KUKA KRL program: MyProgram_037().src

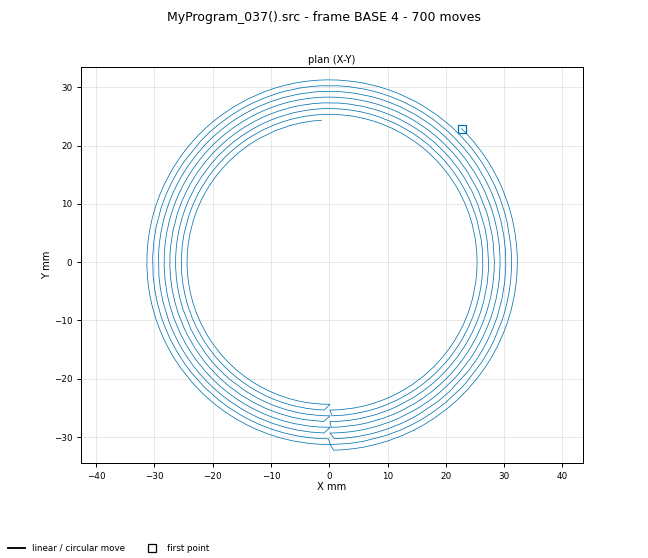
[picture p0: tool path of MyProgram_037().src in frame BASE 4, 700 of 700 moves have a stored position in this frame; points joined in program order, loops and branches not executed]
&ACCESS RVP
&REL 1
&PARAM TEMPLATE = C:\KRC\Roboter\Template\vorgabe
&PARAM EDITMASK = *
DEF MyProgram_037()
; ---- Setting reference (Base) ----
$BASE = BASE_DATA[4]

; --------------------------
; ---- Setting tool (TCP) ----
$TOOL = TOOL_DATA[3]
; --------------------------

$VEL.CP = VEL_APROX_PRINT
Startdeposition()
$VEL.CP = VEL_PRINT
LIN {X 22.7221,Y 22.9099,Z 61,A 36.8926,B 24.82,C -3.0943,E1 25.1146,E2 -314.0122} C_DIS
LIN {X 23.9604,Y 21.6116,Z 61,A 34.1206,B 24.8202,C -3.0927,E1 25.1199,E2 -311.2486} C_DIS
LIN {X 24.912,Y 20.5075,Z 61,A 31.2026,B 24.8214,C -3.0826,E1 25.1251,E2 -308.3199} C_DIS
LIN {X 26.1407,Y 18.916,Z 61,A 27.904,B 24.8219,C -3.0777,E1 25.1306,E2 -305.0254} C_DIS
LIN {X 27.166,Y 17.4114,Z 61,A 24.6548,B 24.8229,C -3.0694,E1 25.1357,E2 -301.7727} C_DIS
LIN {X 28.0132,Y 16.0124,Z 61,A 21.6335,B 24.8239,C -3.0603,E1 25.1399,E2 -298.7454} C_DIS
LIN {X 29.0213,Y 14.1043,Z 61,A 17.6844,B 24.8253,C -3.0484,E1 25.1449,E2 -294.7892} C_DIS
LIN {X 29.7593,Y 12.4714,Z 61,A 14.5862,B 24.8262,C -3.0407,E1 25.1484,E2 -291.6895} C_DIS
LIN {X 30.8171,Y 9.5631,Z 61,A 8.5757,B 24.8288,C -3.0179,E1 25.1538,E2 -285.6589} C_DIS
LIN {X 31.4239,Y 7.3275,Z 61,A 5.4377,B 24.8287,C -3.0189,E1 25.1559,E2 -282.5414} C_DIS
LIN {X 31.8366,Y 5.2519,Z 61,A 0.8875,B 24.8312,C -2.9966,E1 25.1582,E2 -277.9651} C_DIS
LIN {X 32.1427,Y 2.8314,Z 61,A -2.7277,B 24.8316,C -2.9931,E1 25.1593,E2 -274.363} C_DIS
LIN {X 32.236,Y 1.4111,Z 61,A -5.1666,B 24.8324,C -2.9865,E1 25.1597,E2 -271.9229} C_DIS
LIN {X 32.266,Y -0.0088,Z 61,A -7.9428,B 24.8337,C -2.9751,E1 25.1597,E2 -269.1363} C_DIS
LIN {X 32.2046,Y -2.0098,Z 61,A -11.4053,B 24.8348,C -2.9652,E1 25.1593,E2 -265.6709} C_DIS
LIN {X 32.0309,Y -3.8974,Z 61,A -14.9413,B 24.8362,C -2.9523,E1 25.1583,E2 -262.1254} C_DIS
LIN {X 31.7367,Y -5.8263,Z 61,A -18.1738,B 24.837,C -2.9447,E1 25.1568,E2 -258.8938} C_DIS
LIN {X 31.2216,Y -8.147,Z 61,A -22.8563,B 24.8392,C -2.9253,E1 25.1537,E2 -254.1926} C_DIS
LIN {X 30.6383,Y -10.1233,Z 61,A -25.8233,B 24.8394,C -2.9237,E1 25.1512,E2 -251.2384} C_DIS
LIN {X 29.8919,Y -12.1501,Z 61,A -30.2718,B 24.8416,C -2.9038,E1 25.1467,E2 -246.7676} C_DIS
LIN {X 28.8147,Y -14.5215,Z 61,A -34.7253,B 24.8428,C -2.8926,E1 25.1414,E2 -242.3116} C_DIS
LIN {X 27.7798,Y -16.4144,Z 61,A -38.242,B 24.8435,C -2.8861,E1 25.1365,E2 -238.7975} C_DIS
LIN {X 26.8232,Y -17.9358,Z 61,A -41.3536,B 24.8443,C -2.8784,E1 25.1318,E2 -235.6833} C_DIS
LIN {X 25.4842,Y -19.7918,Z 61,A -45.8741,B 24.8462,C -2.8616,E1 25.1242,E2 -231.1447} C_DIS
LIN {X 23.7816,Y -21.8079,Z 61,A -50.4062,B 24.8472,C -2.8519,E1 25.1158,E2 -226.61} C_DIS
LIN {X 22.0503,Y -23.5572,Z 61,A -54.7017,B 24.8482,C -2.8426,E1 25.1072,E2 -222.3105} C_DIS
LIN {X 20.232,Y -25.1362,Z 61,A -58.9185,B 24.8491,C -2.8341,E1 25.0982,E2 -218.0897} C_DIS
LIN {X 18.0334,Y -26.7573,Z 61,A -64.2333,B 24.8508,C -2.8186,E1 25.086,E2 -212.7565} C_DIS
LIN {X 16.0936,Y -27.9669,Z 61,A -67.2597,B 24.8502,C -2.8242,E1 25.0788,E2 -209.7528} C_DIS
LIN {X 14.6043,Y -28.7727,Z 61,A -70.6753,B 24.8512,C -2.8141,E1 25.0703,E2 -206.3229} C_DIS
LIN {X 12.6886,Y -29.6677,Z 61,A -74.4308,B 24.8518,C -2.8085,E1 25.0608,E2 -202.5634} C_DIS
LIN {X 10.2156,Y -30.6072,Z 61,A -79.763,B 24.8532,C -2.7951,E1 25.0467,E2 -197.2101} C_DIS
LIN {X 7.7675,Y -31.3182,Z 61,A -83.5174,B 24.8528,C -2.7994,E1 25.0366,E2 -193.472} C_DIS
LIN {X 6.0925,Y -31.6861,Z 61,A -86.5057,B 24.853,C -2.7975,E1 25.0284,E2 -190.4828} C_DIS
LIN {X 4.35,Y -31.9726,Z 61,A -89.6463,B 24.8532,C -2.7953,E1 25.0197,E2 -187.3398} C_DIS
LIN {X 2.5855,Y -32.1631,Z 61,A -92.4941,B 24.853,C -2.797,E1 25.0118,E2 -184.4979} C_DIS
LIN {X 0.7515,Y -32.2571,Z 61,A -95.8832,B 24.8533,C -2.7944,E1 25.0024,E2 -181.1037} C_DIS
LIN {X 0.7515,Y -32.2571,Z 61,A -95.8832,B 24.8533,C -2.7944,E1 25.0024,E2 -181.1037} C_DIS
Enddeposition()
LIN {X 0.1793,Y -31.277,Z 61,A -95.2426,B 24.8496,C -2.8293,E1 25.0044,E2 -181.8273} C_DIS
Startdeposition()
$VEL.CP = VEL_PRINT
LIN {X 3.3211,Y -31.1043,Z 61,A -89.5129,B 24.8494,C -2.8315,E1 25.0204,E2 -187.5594} C_DIS
LIN {X 5.8203,Y -30.7348,Z 61,A -84.3877,B 24.8484,C -2.8408,E1 25.0345,E2 -192.7011} C_DIS
LIN {X 9.7861,Y -29.7112,Z 61,A -76.8094,B 24.8474,C -2.8498,E1 25.0548,E2 -200.288} C_DIS
LIN {X 12.2324,Y -28.7911,Z 61,A -73.017,B 24.848,C -2.8443,E1 25.0646,E2 -204.0588} C_DIS
LIN {X 13.9421,Y -28.0031,Z 61,A -69.1318,B 24.8469,C -2.855,E1 25.0744,E2 -207.9593} C_DIS
LIN {X 15.7865,Y -27.0066,Z 61,A -66.0402,B 24.8471,C -2.8524,E1 25.0819,E2 -211.0355} C_DIS
LIN {X 17.661,Y -25.8198,Z 61,A -60.7635,B 24.8447,C -2.8754,E1 25.0943,E2 -216.3493} C_DIS
LIN {X 19.9043,Y -24.1326,Z 61,A -55.5619,B 24.8434,C -2.8872,E1 25.1057,E2 -221.5593} C_DIS
LIN {X 22.7108,Y -21.5119,Z 61,A -49.7962,B 24.8434,C -2.887,E1 25.1171,E2 -227.3007} C_DIS
LIN {X 23.4756,Y -20.6753,Z 61,A -46.3418,B 24.8408,C -2.9105,E1 25.1236,E2 -230.795} C_DIS
LIN {X 26.1964,Y -17.0974,Z 61,A -38.73,B 24.8393,C -2.924,E1 25.1359,E2 -238.4019} C_DIS
LIN {X 27.5194,Y -14.8741,Z 61,A -34.5181,B 24.8386,C -2.9303,E1 25.1417,E2 -242.6068} C_DIS
LIN {X 28.3302,Y -13.2648,Z 61,A -30.4988,B 24.8365,C -2.9497,E1 25.1466,E2 -246.6505} C_DIS
LIN {X 29.6792,Y -9.8843,Z 61,A -24.9159,B 24.8359,C -2.9548,E1 25.1521,E2 -252.2145} C_DIS
LIN {X 30.0713,Y -8.6185,Z 61,A -22.3462,B 24.8349,C -2.9642,E1 25.1541,E2 -254.7917} C_DIS
LIN {X 30.4929,Y -6.9814,Z 61,A -19.0418,B 24.8335,C -2.9766,E1 25.1563,E2 -258.1064} C_DIS
LIN {X 30.8584,Y -5.1295,Z 61,A -15.6608,B 24.8324,C -2.9864,E1 25.158,E2 -261.4906} C_DIS
LIN {X 31.1322,Y -3.0618,Z 61,A -11.7675,B 24.8309,C -2.9993,E1 25.1593,E2 -265.3916} C_DIS
LIN {X 31.2639,Y -1.0643,Z 61,A -8.2104,B 24.8298,C -3.0093,E1 25.1597,E2 -268.9512} C_DIS
LIN {X 31.2659,Y 0.9986,Z 61,A -4.0775,B 24.8279,C -3.026,E1 25.1595,E2 -273.099} C_DIS
LIN {X 31.1526,Y 2.8404,Z 61,A -0.0947,B 24.8257,C -3.0448,E1 25.1585,E2 -277.1027} C_DIS
LIN {X 30.502,Y 6.9419,Z 61,A 6.4981,B 24.8247,C -3.0539,E1 25.1552,E2 -283.6785} C_DIS
LIN {X 30.1115,Y 8.4753,Z 61,A 9.5892,B 24.8234,C -3.0651,E1 25.1529,E2 -286.7783} C_DIS
LIN {X 29.2983,Y 10.9626,Z 61,A 13.7921,B 24.8227,C -3.0709,E1 25.1491,E2 -290.9715} C_DIS
LIN {X 28.4168,Y 13.078,Z 61,A 18.7309,B 24.8202,C -3.0925,E1 25.1436,E2 -295.9345} C_DIS
LIN {X 27.2863,Y 15.2975,Z 61,A 22.9812,B 24.8193,C -3.1005,E1 25.138,E2 -300.1813} C_DIS
LIN {X 26.2057,Y 17.0833,Z 61,A 26.3044,B 24.8189,C -3.1036,E1 25.1331,E2 -303.4952} C_DIS
LIN {X 25.2575,Y 18.4557,Z 61,A 29.3022,B 24.8181,C -3.1103,E1 25.1282,E2 -306.4942} C_DIS
LIN {X 24.5119,Y 19.4351,Z 61,A 31.6052,B 24.8174,C -3.1163,E1 25.1243,E2 -308.8004} C_DIS
LIN {X 23.7173,Y 20.3976,Z 61,A 34.2425,B 24.8163,C -3.1259,E1 25.1195,E2 -311.4486} C_DIS
LIN {X 22.3374,Y 21.899,Z 61,A 37.6321,B 24.8159,C -3.1295,E1 25.113,E2 -314.8319} C_DIS
LIN {X 21.2569,Y 22.9504,Z 61,A 40.4087,B 24.8152,C -3.1352,E1 25.1074,E2 -317.6107} C_DIS
LIN {X 20.2008,Y 23.8849,Z 61,A 43.3561,B 24.8141,C -3.1446,E1 25.1011,E2 -320.5688} C_DIS
LIN {X 18.523,Y 25.2082,Z 61,A 47.5292,B 24.8129,C -3.1545,E1 25.0918,E2 -324.7504} C_DIS
LIN {X 15.977,Y 26.894,Z 61,A 52.4422,B 24.8129,C -3.1548,E1 25.0803,E2 -329.6481} C_DIS
LIN {X 14.9451,Y 27.4809,Z 61,A 55.3612,B 24.8115,C -3.1665,E1 25.0731,E2 -332.5865} C_DIS
LIN {X 12.1463,Y 28.8274,Z 61,A 60.2984,B 24.8117,C -3.1641,E1 25.0606,E2 -337.5056} C_DIS
LIN {X 10.3203,Y 29.5304,Z 61,A 64.2509,B 24.8109,C -3.1715,E1 25.0502,E2 -341.4674} C_DIS
LIN {X 8.4349,Y 30.123,Z 61,A 68.0075,B 24.8104,C -3.1755,E1 25.0401,E2 -345.2271} C_DIS
LIN {X 5.8555,Y 30.729,Z 61,A 72.4111,B 24.8107,C -3.1729,E1 25.0281,E2 -349.6186} C_DIS
LIN {X 4.2839,Y 30.987,Z 61,A 75.855,B 24.8099,C -3.1793,E1 25.0186,E2 -353.0747} C_DIS
LIN {X 1.5654,Y 31.243,Z 61,A 80.5109,B 24.8103,C -3.1759,E1 25.0057,E2 -357.7202} C_DIS
LIN {X -0.4527,Y 31.2782,Z 61,A 83.939,B 24.8107,C -3.1724,E1 24.9961,E2 -361.14} C_DIS
LIN {X -1.9504,Y 31.2214,Z 61,A 86.8625,B 24.8107,C -3.1733,E1 24.988,E2 -364.0661} C_DIS
LIN {X -3.7004,Y 31.0622,Z 61,A 89.7933,B 24.8112,C -3.1688,E1 24.9798,E2 -366.9879} C_DIS
LIN {X -4.8807,Y 30.8989,Z 61,A 92.0557,B 24.8112,C -3.1681,E1 24.9736,E2 -369.2507} C_DIS
LIN {X -6.0959,Y 30.6823,Z 61,A 94.5824,B 24.8112,C -3.1689,E1 24.9666,E2 -371.7821} C_DIS
LIN {X -7.8851,Y 30.2715,Z 61,A 97.7613,B 24.8117,C -3.1641,E1 24.958,E2 -374.9538} C_DIS
LIN {X -9.34,Y 29.855,Z 61,A 100.6774,B 24.8119,C -3.1624,E1 24.9502,E2 -377.8709} C_DIS
LIN {X -10.9576,Y 29.3002,Z 61,A 104.3444,B 24.8119,C -3.1635,E1 24.9406,E2 -381.5478} C_DIS
LIN {X -13.786,Y 28.0804,Z 61,A 109.2809,B 24.8136,C -3.1489,E1 24.9281,E2 -386.4614} C_DIS
LIN {X -16.3147,Y 26.6903,Z 61,A 115.7502,B 24.8134,C -3.1501,E1 24.9124,E2 -392.9529} C_DIS
LIN {X -18.6587,Y 25.1078,Z 61,A 120.0777,B 24.8155,C -3.1326,E1 24.9026,E2 -397.2535} C_DIS
LIN {X -20.009,Y 24.0456,Z 61,A 123.0586,B 24.8164,C -3.1246,E1 24.8962,E2 -400.2265} C_DIS
LIN {X -21.1218,Y 23.0743,Z 61,A 125.7069,B 24.8172,C -3.1181,E1 24.8907,E2 -402.8698} C_DIS
LIN {X -22.43,Y 21.8051,Z 61,A 129.3952,B 24.8178,C -3.1131,E1 24.8834,E2 -406.5617} C_DIS
LIN {X -24.1295,Y 19.9081,Z 61,A 134.5719,B 24.8187,C -3.1056,E1 24.874,E2 -411.7439} C_DIS
LIN {X -25.5591,Y 18.0363,Z 61,A 138.1819,B 24.8206,C -3.0887,E1 24.868,E2 -415.331} C_DIS
LIN {X -26.9094,Y 15.9512,Z 61,A 143.7462,B 24.8212,C -3.084,E1 24.8598,E2 -420.9126} C_DIS
LIN {X -28.2304,Y 13.4761,Z 61,A 148.1193,B 24.8236,C -3.0633,E1 24.8544,E2 -425.2597} C_DIS
LIN {X -29.0622,Y 11.5738,Z 61,A 151.9664,B 24.8249,C -3.0524,E1 24.8502,E2 -429.102} C_DIS
LIN {X -29.7747,Y 9.5928,Z 61,A 156.0479,B 24.826,C -3.0425,E1 24.8466,E2 -433.1829} C_DIS
LIN {X -30.3453,Y 7.5996,Z 61,A 159.7045,B 24.8275,C -3.0298,E1 24.844,E2 -436.8303} C_DIS
LIN {X -30.7795,Y 5.5835,Z 61,A 163.4375,B 24.8288,C -3.0178,E1 24.8419,E2 -440.5566} C_DIS
LIN {X -31.0699,Y 3.635,Z 61,A 167.201,B 24.83,C -3.0076,E1 24.8406,E2 -444.3184} C_DIS
LIN {X -31.2361,Y 1.691,Z 61,A 170.4385,B 24.8315,C -2.994,E1 24.8399,E2 -447.5426} C_DIS
LIN {X -31.2747,Y -0.673,Z 61,A 175.5679,B 24.8324,C -2.9864,E1 24.8399,E2 -452.6848} C_DIS
LIN {X -31.1425,Y -2.9504,Z 61,A 179.1206,B 24.8344,C -2.9688,E1 24.8407,E2 -456.2167} C_DIS
LIN {X -30.9732,Y -4.3828,Z 61,A -178.3923,B 24.8354,C -2.9596,E1 24.8416,E2 -458.6965} C_DIS
LIN {X -30.7489,Y -5.7508,Z 61,A -175.6308,B 24.8361,C -2.9535,E1 24.8429,E2 -461.4599} C_DIS
LIN {X -30.3552,Y -7.5574,Z 61,A -172.6642,B 24.8375,C -2.9402,E1 24.8448,E2 -464.4121} C_DIS
LIN {X -29.7953,Y -9.529,Z 61,A -167.6721,B 24.8377,C -2.9386,E1 24.8488,E2 -469.4292} C_DIS
LIN {X -29.0107,Y -11.7023,Z 61,A -164.0836,B 24.8396,C -2.9217,E1 24.8524,E2 -472.9972} C_DIS
LIN {X -28.2977,Y -13.333,Z 61,A -160.8621,B 24.8406,C -2.9124,E1 24.8561,E2 -476.2141} C_DIS
LIN {X -27.3621,Y -15.1617,Z 61,A -157.5041,B 24.8421,C -2.8992,E1 24.8605,E2 -479.5584} C_DIS
LIN {X -26.5372,Y -16.5628,Z 61,A -153.809,B 24.8423,C -2.8973,E1 24.8659,E2 -483.2679} C_DIS
LIN {X -25.4676,Y -18.1646,Z 61,A -149.9018,B 24.8429,C -2.8918,E1 24.8721,E2 -487.1813} C_DIS
LIN {X -23.4143,Y -20.7446,Z 61,A -144.5543,B 24.845,C -2.8724,E1 24.8816,E2 -492.5069} C_DIS
LIN {X -21.7484,Y -22.4847,Z 61,A -139.595,B 24.8455,C -2.8679,E1 24.8914,E2 -497.4768} C_DIS
LIN {X -19.7938,Y -24.2225,Z 61,A -134.708,B 24.8463,C -2.8599,E1 24.9018,E2 -502.3635} C_DIS
LIN {X -17.9022,Y -25.6528,Z 61,A -131.385,B 24.8481,C -2.8435,E1 24.9092,E2 -505.6591} C_DIS
LIN {X -16.1813,Y -26.7715,Z 61,A -126.5019,B 24.8476,C -2.8482,E1 24.9208,E2 -510.5689} C_DIS
LIN {X -14.1331,Y -27.9074,Z 61,A -122.7805,B 24.8487,C -2.8375,E1 24.9299,E2 -514.275} C_DIS
LIN {X -12.3744,Y -28.7304,Z 61,A -119.0798,B 24.849,C -2.835,E1 24.9394,E2 -517.9789} C_DIS
LIN {X -10.1671,Y -29.5837,Z 61,A -114.3689,B 24.849,C -2.835,E1 24.9518,E2 -522.6992} C_DIS
LIN {X -8.2154,Y -30.1838,Z 61,A -111.3645,B 24.8501,C -2.8252,E1 24.9598,E2 -525.6852} C_DIS
LIN {X -6.0483,Y -30.6918,Z 61,A -106.3449,B 24.8492,C -2.8331,E1 24.9735,E2 -530.7296} C_DIS
LIN {X -3.3817,Y -31.0983,Z 61,A -101.8901,B 24.8499,C -2.8271,E1 24.9858,E2 -535.1734} C_DIS
LIN {X -1.2466,Y -31.2571,Z 61,A -97.8183,B 24.8497,C -2.8289,E1 24.9972,E2 -539.2508} C_DIS
LIN {X 0.1793,Y -31.277,Z 61,A -95.2424,B 24.8497,C -2.8292,E1 25.0044,E2 -541.8272} C_DIS
Enddeposition()
LIN {X 0.1793,Y -31.277,Z 61,A -95.2424,B 24.8497,C -2.8292,E1 25.0044,E2 -541.8272} C_DIS
Startdeposition()
$VEL.CP = VEL_PRINT
LIN {X -0.1083,Y -30.2967,Z 61,A -97.7907,B 24.8501,C -2.8248,E1 24.9973,E2 -539.2685} C_DIS
LIN {X -1.7664,Y -30.2454,Z 61,A -100.7174,B 24.8499,C -2.8266,E1 24.9891,E2 -536.3455} C_DIS
LIN {X -3.5776,Y -30.0849,Z 61,A -104.4761,B 24.8502,C -2.8238,E1 24.9786,E2 -532.5779} C_DIS
LIN {X -5.7242,Y -29.7511,Z 61,A -108.6372,B 24.8502,C -2.8245,E1 24.9672,E2 -528.4145} C_DIS
LIN {X -7.9,Y -29.2487,Z 61,A -112.9088,B 24.8499,C -2.8264,E1 24.9556,E2 -524.1412} C_DIS
LIN {X -9.8571,Y -28.6489,Z 61,A -116.5327,B 24.8494,C -2.8315,E1 24.946,E2 -520.523} C_DIS
LIN {X -12.0715,Y -27.7881,Z 61,A -121.794,B 24.8496,C -2.8291,E1 24.9324,E2 -515.2441} C_DIS
LIN {X -14.1119,Y -26.8095,Z 61,A -125.1264,B 24.8482,C -2.8425,E1 24.9241,E2 -511.9348} C_DIS
LIN {X -15.2026,Y -26.2056,Z 61,A -127.7329,B 24.8481,C -2.8436,E1 24.9178,E2 -509.3231} C_DIS
LIN {X -17.2127,Y -24.9324,Z 61,A -132.0881,B 24.8472,C -2.8516,E1 24.9076,E2 -504.973} C_DIS
LIN {X -18.9208,Y -23.6626,Z 61,A -136.9417,B 24.8472,C -2.8518,E1 24.8969,E2 -500.1021} C_DIS
LIN {X -21.3596,Y -21.4865,Z 61,A -143.2342,B 24.846,C -2.8632,E1 24.8841,E2 -493.811} C_DIS
LIN {X -23.5988,Y -19.0001,Z 61,A -149.3266,B 24.8443,C -2.8791,E1 24.8731,E2 -487.729} C_DIS
LIN {X -24.7571,Y -17.4644,Z 61,A -152.8937,B 24.8432,C -2.8884,E1 24.8672,E2 -484.1666} C_DIS
LIN {X -26.1364,Y -15.323,Z 61,A -157.5379,B 24.8418,C -2.9019,E1 24.8604,E2 -479.5311} C_DIS
LIN {X -27.4184,Y -12.8894,Z 61,A -163.2384,B 24.8406,C -2.9124,E1 24.8533,E2 -473.8249} C_DIS
LIN {X -28.2493,Y -10.9495,Z 61,A -166.6876,B 24.839,C -2.9274,E1 24.8497,E2 -470.3925} C_DIS
LIN {X -28.8492,Y -9.2519,Z 61,A -170.1049,B 24.8379,C -2.9372,E1 24.8467,E2 -466.979} C_DIS
LIN {X -29.4938,Y -6.9298,Z 61,A -174.3156,B 24.8361,C -2.9531,E1 24.8437,E2 -462.7818} C_DIS
LIN {X -29.9388,Y -4.644,Z 61,A -179.87,B 24.8355,C -2.9587,E1 24.841,E2 -457.2079} C_DIS
LIN {X -30.1985,Y -2.439,Z 61,A 175.975,B 24.834,C -2.9719,E1 24.84,E2 -453.0596} C_DIS
LIN {X -30.2834,Y 0.8875,Z 61,A 170.1741,B 24.8314,C -2.9948,E1 24.84,E2 -447.2787} C_DIS
LIN {X -30.0832,Y 3.5884,Z 61,A 164.9418,B 24.8297,C -3.0101,E1 24.8413,E2 -442.0516} C_DIS
LIN {X -29.6827,Y 6.0689,Z 61,A 159.6211,B 24.8284,C -3.0211,E1 24.844,E2 -436.7256} C_DIS
LIN {X -28.8326,Y 9.3041,Z 61,A 153.6942,B 24.8259,C -3.0431,E1 24.8486,E2 -430.8171} C_DIS
LIN {X -28.0084,Y 11.5504,Z 61,A 149.1158,B 24.8244,C -3.0562,E1 24.8533,E2 -426.2445} C_DIS
LIN {X -27.0518,Y 13.6423,Z 61,A 145.6235,B 24.8223,C -3.0748,E1 24.8574,E2 -422.7777} C_DIS
LIN {X -26.0575,Y 15.4565,Z 61,A 140.2107,B 24.8223,C -3.0753,E1 24.8649,E2 -417.3379} C_DIS
LIN {X -24.8873,Y 17.2777,Z 61,A 135.6577,B 24.8213,C -3.083,E1 24.8722,E2 -412.781} C_DIS
LIN {X -21.994,Y 20.8368,Z 61,A 128.3614,B 24.8176,C -3.1147,E1 24.8854,E2 -405.5272} C_DIS
LIN {X -20.6237,Y 22.1937,Z 61,A 124.5732,B 24.8167,C -3.122,E1 24.893,E2 -401.7408} C_DIS
LIN {X -19.0927,Y 23.5236,Z 61,A 120.2867,B 24.8162,C -3.1268,E1 24.9022,E2 -397.4494} C_DIS
LIN {X -17.0972,Y 25.0118,Z 61,A 116.1796,B 24.8145,C -3.1408,E1 24.9115,E2 -393.3615} C_DIS
LIN {X -15.5028,Y 26.0301,Z 61,A 112.0706,B 24.8143,C -3.143,E1 24.9212,E2 -389.2449} C_DIS
LIN {X -13.5594,Y 27.0934,Z 61,A 107.8903,B 24.8134,C -3.1498,E1 24.9316,E2 -385.0695} C_DIS
LIN {X -11.1624,Y 28.1657,Z 61,A 102.7878,B 24.8128,C -3.1556,E1 24.9447,E2 -379.969} C_DIS
LIN {X -8.6144,Y 29.0463,Z 61,A 98.1678,B 24.8116,C -3.1656,E1 24.9569,E2 -375.3644} C_DIS
LIN {X -7.4328,Y 29.3704,Z 61,A 95.5053,B 24.8116,C -3.1647,E1 24.9642,E2 -372.6961} C_DIS
LIN {X -5.0851,Y 29.8671,Z 61,A 91.1536,B 24.811,C -3.1699,E1 24.9761,E2 -368.3521} C_DIS
LIN {X -2.8898,Y 30.1588,Z 61,A 86.9107,B 24.8108,C -3.1717,E1 24.9878,E2 -364.1107} C_DIS
LIN {X -1.489,Y 30.2599,Z 61,A 83.7084,B 24.8113,C -3.1675,E1 24.9968,E2 -360.8976} C_DIS
LIN {X 1.7595,Y 30.2458,Z 61,A 78.3913,B 24.8103,C -3.1762,E1 25.0116,E2 -355.6022} C_DIS
LIN {X 3.3881,Y 30.1066,Z 61,A 74.7935,B 24.8109,C -3.1708,E1 25.0216,E2 -351.9938} C_DIS
LIN {X 6.0588,Y 29.6848,Z 61,A 70.2105,B 24.8105,C -3.1744,E1 25.0342,E2 -347.4243} C_DIS
LIN {X 7.6214,Y 29.3225,Z 61,A 67.3022,B 24.8105,C -3.1741,E1 25.042,E2 -344.5194} C_DIS
LIN {X 8.8433,Y 28.9774,Z 61,A 64.8089,B 24.8109,C -3.1714,E1 25.0487,E2 -342.0241} C_DIS
LIN {X 10.5374,Y 28.4057,Z 61,A 61.2512,B 24.8114,C -3.1666,E1 25.0581,E2 -338.4622} C_DIS
LIN {X 12.6517,Y 27.5291,Z 61,A 56.5705,B 24.8124,C -3.1582,E1 25.0701,E2 -333.7727} C_DIS
LIN {X 14.7691,Y 26.4532,Z 61,A 52.4965,B 24.8126,C -3.157,E1 25.0801,E2 -329.7076} C_DIS
LIN {X 15.97,Y 25.7457,Z 61,A 49.6207,B 24.8134,C -3.1505,E1 25.087,E2 -326.8252} C_DIS
LIN {X 17.8127,Y 24.5075,Z 61,A 45.2964,B 24.8144,C -3.1422,E1 25.0969,E2 -322.4961} C_DIS
LIN {X 19.9808,Y 22.7742,Z 61,A 40.5699,B 24.8148,C -3.1387,E1 25.107,E2 -317.7793} C_DIS
LIN {X 21.1552,Y 21.687,Z 61,A 37.0416,B 24.8162,C -3.1266,E1 25.1142,E2 -314.2371} C_DIS
LIN {X 23.0143,Y 19.7039,Z 61,A 32.585,B 24.8165,C -3.1237,E1 25.1225,E2 -309.7933} C_DIS
LIN {X 24.2227,Y 18.1978,Z 61,A 28.2223,B 24.8186,C -3.1064,E1 25.13,E2 -305.4102} C_DIS
LIN {X 25.3541,Y 16.5854,Z 61,A 24.1344,B 24.8202,C -3.0927,E1 25.1363,E2 -301.3101} C_DIS
LIN {X 27.0232,Y 13.6987,Z 61,A 18.5921,B 24.821,C -3.0856,E1 25.1438,E2 -295.78} C_DIS
LIN {X 27.9171,Y 11.7698,Z 61,A 14.7622,B 24.822,C -3.0769,E1 25.1481,E2 -291.9502} C_DIS
LIN {X 28.5269,Y 10.2035,Z 61,A 10.9832,B 24.824,C -3.0601,E1 25.1518,E2 -288.1527} C_DIS
LIN {X 29.4353,Y 7.1737,Z 61,A 5.6519,B 24.825,C -3.0508,E1 25.1558,E2 -282.83} C_DIS
LIN {X 29.9505,Y 4.5682,Z 61,A -0.1932,B 24.828,C -3.0249,E1 25.1586,E2 -276.9578} C_DIS
LIN {X 30.2349,Y 1.9385,Z 61,A -4.6467,B 24.829,C -3.0166,E1 25.1596,E2 -272.5109} C_DIS
LIN {X 30.2949,Y -0.3425,Z 61,A -8.9772,B 24.8305,C -3.0029,E1 25.1596,E2 -268.1738} C_DIS
LIN {X 30.124,Y -3.2324,Z 61,A -14.8109,B 24.833,C -2.9811,E1 25.1583,E2 -262.323} C_DIS
LIN {X 29.6574,Y -6.1925,Z 61,A -20.1219,B 24.8344,C -2.9681,E1 25.1557,E2 -257.0124} C_DIS
LIN {X 28.8629,Y -9.211,Z 61,A -24.9574,B 24.8349,C -2.964,E1 25.1521,E2 -252.1948} C_DIS
LIN {X 28.0924,Y -11.3454,Z 61,A -30.7262,B 24.8385,C -2.9319,E1 25.1463,E2 -246.3822} C_DIS
LIN {X 27.0866,Y -13.5732,Z 61,A -34.1792,B 24.8383,C -2.9335,E1 25.1422,E2 -242.9516} C_DIS
LIN {X 26.3833,Y -14.8943,Z 61,A -37.27,B 24.8396,C -2.9221,E1 25.138,E2 -239.8499} C_DIS
LIN {X 25.3403,Y -16.6064,Z 61,A -40.3805,B 24.8397,C -2.9203,E1 25.1334,E2 -236.7509} C_DIS
LIN {X 23.953,Y -18.5514,Z 61,A -46.8407,B 24.8437,C -2.8839,E1 25.1226,E2 -230.2355} C_DIS
LIN {X 20.6747,Y -22.1465,Z 61,A -55.9829,B 24.846,C -2.8628,E1 25.1046,E2 -221.0822} C_DIS
LIN {X 18.623,Y -23.8975,Z 61,A -60.9233,B 24.847,C -2.8539,E1 25.0938,E2 -216.1391} C_DIS
LIN {X 15.2202,Y -26.1966,Z 61,A -67.5031,B 24.847,C -2.8534,E1 25.0784,E2 -209.5794} C_DIS
LIN {X 13.4821,Y -27.1315,Z 61,A -70.9533,B 24.8473,C -2.8506,E1 25.0699,E2 -206.1321} C_DIS
LIN {X 12.1806,Y -27.7404,Z 61,A -73.8495,B 24.848,C -2.8444,E1 25.0625,E2 -203.2286} C_DIS
LIN {X 10.1217,Y -28.5562,Z 61,A -78.4977,B 24.8491,C -2.8337,E1 25.0503,E2 -198.5649} C_DIS
LIN {X 8.3465,Y -29.1245,Z 61,A -81.7097,B 24.8491,C -2.8333,E1 25.0417,E2 -195.3574} C_DIS
LIN {X 6.916,Y -29.4969,Z 61,A -84.6101,B 24.8496,C -2.8295,E1 25.0338,E2 -192.4522} C_DIS
LIN {X 4.7564,Y -29.9211,Z 61,A -88.6328,B 24.8498,C -2.8278,E1 25.0228,E2 -188.4297} C_DIS
LIN {X 2.5826,Y -30.186,Z 61,A -92.4841,B 24.8498,C -2.8285,E1 25.0121,E2 -184.5828} C_DIS
LIN {X 0.8989,Y -30.2834,Z 61,A -95.9394,B 24.8501,C -2.8246,E1 25.0024,E2 -181.1192} C_DIS
LIN {X 0.8989,Y -30.2834,Z 61,A -95.9394,B 24.8501,C -2.8246,E1 25.0024,E2 -181.1192} C_DIS
Enddeposition()
LIN {X 0.148,Y -29.3098,Z 61,A -95.712,B 24.8465,C -2.8581,E1 25.0033,E2 -181.4265} C_DIS
Startdeposition()
$VEL.CP = VEL_PRINT
LIN {X 2.0107,Y -29.2427,Z 61,A -92.0588,B 24.8464,C -2.8596,E1 25.0135,E2 -185.0819} C_DIS
LIN {X 3.7148,Y -29.075,Z 61,A -88.9657,B 24.8464,C -2.8588,E1 25.022,E2 -188.171} C_DIS
LIN {X 4.9608,Y -28.8892,Z 61,A -86.4055,B 24.8461,C -2.8616,E1 25.0291,E2 -190.7354} C_DIS
LIN {X 6.1622,Y -28.6568,Z 61,A -83.7025,B 24.8456,C -2.8671,E1 25.0365,E2 -193.4479} C_DIS
LIN {X 7.9763,Y -28.2057,Z 61,A -79.7952,B 24.8448,C -2.8736,E1 25.0471,E2 -197.3645} C_DIS
LIN {X 10.4914,Y -27.3695,Z 61,A -75.5865,B 24.8453,C -2.8692,E1 25.0581,E2 -201.5543} C_DIS
LIN {X 11.7916,Y -26.8355,Z 61,A -71.1886,B 24.8428,C -2.8921,E1 25.0695,E2 -205.9959} C_DIS
LIN {X 15.0472,Y -25.1549,Z 61,A -64.7391,B 24.8424,C -2.8959,E1 25.0853,E2 -212.4357} C_DIS
LIN {X 17.2957,Y -23.6651,Z 61,A -59.7421,B 24.8417,C -2.9029,E1 25.0967,E2 -217.4323} C_DIS
LIN {X 18.7666,Y -22.5166,Z 61,A -55.493,B 24.84,C -2.9181,E1 25.1059,E2 -221.7013} C_DIS
LIN {X 21.1943,Y -20.2484,Z 61,A -49.8511,B 24.8395,C -2.9227,E1 25.1172,E2 -227.3306} C_DIS
LIN {X 22.3114,Y -19.01,Z 61,A -45.9121,B 24.8376,C -2.9394,E1 25.1244,E2 -231.2913} C_DIS
LIN {X 24.1424,Y -16.623,Z 61,A -40.9595,B 24.8372,C -2.9432,E1 25.1326,E2 -236.2291} C_DIS
LIN {X 24.8001,Y -15.6252,Z 61,A -38.3769,B 24.8361,C -2.9528,E1 25.1365,E2 -238.8214} C_DIS
LIN {X 25.6751,Y -14.1403,Z 61,A -35.035,B 24.8351,C -2.962,E1 25.1412,E2 -242.1677} C_DIS
LIN {X 26.337,Y -12.8674,Z 61,A -32.0159,B 24.8339,C -2.9728,E1 25.1449,E2 -245.1965} C_DIS
LIN {X 27.1667,Y -11.006,Z 61,A -28.3627,B 24.8331,C -2.9804,E1 25.1489,E2 -248.8475} C_DIS
LIN {X 27.762,Y -9.4049,Z 61,A -25.2808,B 24.8323,C -2.9871,E1 25.1518,E2 -251.928} C_DIS
LIN {X 28.1054,Y -8.3226,Z 61,A -22.5879,B 24.8308,C -3,E1 25.154,E2 -254.6362} C_DIS
LIN {X 28.6095,Y -6.377,Z 61,A -18.7112,B 24.8295,C -3.0115,E1 25.1566,E2 -258.5176} C_DIS
LIN {X 29.0038,Y -4.2385,Z 61,A -14.659,B 24.8283,C -3.0221,E1 25.1584,E2 -262.5712} C_DIS
LIN {X 29.2053,Y -2.5002,Z 61,A -11.0811,B 24.8269,C -3.0349,E1 25.1594,E2 -266.1581} C_DIS
LIN {X 29.3074,Y -0.5096,Z 61,A -7.4417,B 24.8259,C -3.0437,E1 25.1598,E2 -269.7969} C_DIS
LIN {X 29.2938,Y 1.0136,Z 61,A -4.2793,B 24.8245,C -3.0554,E1 25.1596,E2 -272.9681} C_DIS
LIN {X 29.1565,Y 3.0136,Z 61,A -0.1704,B 24.8228,C -3.07,E1 25.1585,E2 -277.0872} C_DIS
LIN {X 28.7926,Y 5.4913,Z 61,A 4.4077,B 24.8216,C -3.0808,E1 25.1565,E2 -281.664} C_DIS
LIN {X 28.3607,Y 7.4071,Z 61,A 8.36,B 24.8201,C -3.0937,E1 25.1538,E2 -285.6241} C_DIS
LIN {X 27.7503,Y 9.4393,Z 61,A 12.7184,B 24.8183,C -3.1085,E1 25.1501,E2 -289.9928} C_DIS
LIN {X 26.7315,Y 12.0254,Z 61,A 17.843,B 24.817,C -3.1198,E1 25.1446,E2 -295.116} C_DIS
LIN {X 25.7605,Y 13.9849,Z 61,A 22.1604,B 24.8156,C -3.1318,E1 25.139,E2 -299.4388} C_DIS
LIN {X 24.9032,Y 15.4594,Z 61,A 25.4232,B 24.8147,C -3.1394,E1 25.1343,E2 -302.7033} C_DIS
LIN {X 23.3109,Y 17.771,Z 61,A 31.399,B 24.8124,C -3.1587,E1 25.1245,E2 -308.6957} C_DIS
LIN {X 22.0327,Y 19.3325,Z 61,A 35.2047,B 24.8115,C -3.1658,E1 25.1175,E2 -312.501} C_DIS
LIN {X 19.9544,Y 21.4716,Z 61,A 40.5781,B 24.8108,C -3.1722,E1 25.1068,E2 -317.8672} C_DIS
LIN {X 18.7812,Y 22.5044,Z 61,A 43.4615,B 24.8103,C -3.1759,E1 25.1007,E2 -320.7482} C_DIS
LIN {X 17.2029,Y 23.7331,Z 61,A 48.0223,B 24.8086,C -3.1901,E1 25.0905,E2 -325.3263} C_DIS
LIN {X 14.7834,Y 25.3107,Z 61,A 53.1705,B 24.8083,C -3.1928,E1 25.0783,E2 -330.4646} C_DIS
LIN {X 12.224,Y 26.6417,Z 61,A 59.3231,B 24.8068,C -3.2053,E1 25.0628,E2 -336.6304} C_DIS
LIN {X 10.0639,Y 27.53,Z 61,A 63.0855,B 24.8073,C -3.2009,E1 25.0531,E2 -340.3741} C_DIS
LIN {X 8.62,Y 28.0157,Z 61,A 66.0319,B 24.8071,C -3.2029,E1 25.0453,E2 -343.3197} C_DIS
LIN {X 7.2419,Y 28.4031,Z 61,A 69.0749,B 24.8066,C -3.2071,E1 25.037,E2 -346.3681} C_DIS
LIN {X 4.3754,Y 28.9836,Z 61,A 75.6585,B 24.8052,C -3.218,E1 25.0189,E2 -352.9705} C_DIS
LIN {X 1.9541,Y 29.2466,Z 61,A 80.06,B 24.8056,C -3.2146,E1 25.0067,E2 -357.3618} C_DIS
LIN {X -1.0986,Y 29.2908,Z 61,A 84.8729,B 24.8071,C -3.2024,E1 24.9933,E2 -362.1452} C_DIS
LIN {X -2.3884,Y 29.2143,Z 61,A 88.7301,B 24.8058,C -3.2137,E1 24.9825,E2 -366.0312} C_DIS
LIN {X -5.287,Y 28.8312,Z 61,A 94.0007,B 24.8067,C -3.2058,E1 24.968,E2 -371.2875} C_DIS
LIN {X -7.8717,Y 28.2351,Z 61,A 98.4478,B 24.8081,C -3.1944,E1 24.956,E2 -375.7138} C_DIS
LIN {X -9.6951,Y 27.662,Z 61,A 102.9371,B 24.8078,C -3.1965,E1 24.9441,E2 -380.2164} C_DIS
LIN {X -11.7985,Y 26.8325,Z 61,A 107.3153,B 24.8086,C -3.1901,E1 24.9328,E2 -384.5892} C_DIS
LIN {X -13.2051,Y 26.1691,Z 61,A 110.229,B 24.8093,C -3.1843,E1 24.9255,E2 -387.4968} C_DIS
LIN {X -14.5874,Y 25.4241,Z 61,A 113.1846,B 24.8101,C -3.1782,E1 24.9183,E2 -390.4463} C_DIS
LIN {X -16.1533,Y 24.4591,Z 61,A 116.5351,B 24.8111,C -3.1696,E1 24.9105,E2 -393.7871} C_DIS
LIN {X -17.2445,Y 23.7026,Z 61,A 119.3609,B 24.8115,C -3.1663,E1 24.904,E2 -396.6148} C_DIS
LIN {X -18.6064,Y 22.6494,Z 61,A 122.6877,B 24.8124,C -3.159,E1 24.8968,E2 -399.9364} C_DIS
LIN {X -19.8933,Y 21.5278,Z 61,A 126.2832,B 24.813,C -3.1535,E1 24.8893,E2 -403.5332} C_DIS
LIN {X -21.0236,Y 20.4255,Z 61,A 128.9791,B 24.8142,C -3.1434,E1 24.884,E2 -406.2163} C_DIS
LIN {X -22.5661,Y 18.707,Z 61,A 134.4985,B 24.8147,C -3.1395,E1 24.8739,E2 -411.7514} C_DIS
LIN {X -24.2,Y 16.5395,Z 61,A 139.2149,B 24.8168,C -3.1212,E1 24.8663,E2 -416.447} C_DIS
LIN {X -25.2893,Y 14.8203,Z 61,A 142.6177,B 24.8186,C -3.1062,E1 24.8613,E2 -419.8313} C_DIS
LIN {X -25.9952,Y 13.5443,Z 61,A 145.8028,B 24.8193,C -3.1004,E1 24.8571,E2 -423.0194} C_DIS
LIN {X -26.7357,Y 12.016,Z 61,A 149.4711,B 24.8201,C -3.0932,E1 24.8528,E2 -426.6903} C_DIS
LIN {X -27.4791,Y 10.2033,Z 61,A 153.4524,B 24.8213,C -3.0828,E1 24.8487,E2 -430.669} C_DIS
LIN {X -28.2106,Y 7.9587,Z 61,A 157.5104,B 24.8234,C -3.065,E1 24.8454,E2 -434.7078} C_DIS
LIN {X -28.5007,Y 6.8482,Z 61,A 160.2093,B 24.8238,C -3.0611,E1 24.8436,E2 -437.4133} C_DIS
LIN {X -28.8888,Y 4.9632,Z 61,A 163.9247,B 24.8252,C -3.0492,E1 24.8417,E2 -441.1219} C_DIS
LIN {X -29.1498,Y 3.0762,Z 61,A 167.7373,B 24.8265,C -3.0381,E1 24.8404,E2 -444.931} C_DIS
LIN {X -29.2744,Y 1.4849,Z 61,A 171.9368,B 24.8268,C -3.0357,E1 24.8398,E2 -449.1499} C_DIS
LIN {X -29.2132,Y -2.4024,Z 61,A 177.9508,B 24.8307,C -3.0013,E1 24.8404,E2 -455.1178} C_DIS
LIN {X -28.9639,Y -4.5028,Z 61,A -176.4517,B 24.831,C -2.9986,E1 24.8426,E2 -460.7422} C_DIS
LIN {X -28.4727,Y -6.9631,Z 61,A -171.5064,B 24.8326,C -2.9842,E1 24.8457,E2 -465.682} C_DIS
LIN {X -27.4842,Y -10.1883,Z 61,A -165.8489,B 24.8355,C -2.9586,E1 24.8507,E2 -471.3104} C_DIS
LIN {X -26.8291,Y -11.8058,Z 61,A -162.3427,B 24.8365,C -2.9497,E1 24.8545,E2 -474.8148} C_DIS
LIN {X -25.9454,Y -13.6388,Z 61,A -158.1341,B 24.8375,C -2.9407,E1 24.8598,E2 -479.0245} C_DIS
LIN {X -25.1041,Y -15.1314,Z 61,A -154.9556,B 24.8386,C -2.9308,E1 24.8642,E2 -482.1957} C_DIS
LIN {X -24.0454,Y -16.7631,Z 61,A -151.5159,B 24.8399,C -2.9187,E1 24.8696,E2 -485.6237} C_DIS
LIN {X -23.3784,Y -17.6815,Z 61,A -149.1023,B 24.8403,C -2.9149,E1 24.8736,E2 -488.0398} C_DIS
LIN {X -22.4576,Y -18.8373,Z 61,A -145.9736,B 24.8409,C -2.9102,E1 24.8791,E2 -491.1717} C_DIS
LIN {X -21.2303,Y -20.2109,Z 61,A -142.4266,B 24.8418,C -2.902,E1 24.8858,E2 -494.7148} C_DIS
LIN {X -20.0469,Y -21.3847,Z 61,A -139.0646,B 24.8424,C -2.8963,E1 24.8926,E2 -498.0772} C_DIS
LIN {X -18.4635,Y -22.7657,Z 61,A -134.8248,B 24.8431,C -2.8898,E1 24.9017,E2 -502.3178} C_DIS
LIN {X -17.1315,Y -23.784,Z 61,A -131.6315,B 24.8438,C -2.8837,E1 24.9088,E2 -505.5076} C_DIS
LIN {X -14.9352,Y -25.2214,Z 61,A -126.2324,B 24.8443,C -2.8784,E1 24.9216,E2 -510.9112} C_DIS
LIN {X -13.5636,Y -25.985,Z 61,A -123.3942,B 24.845,C -2.8725,E1 24.9286,E2 -513.7433} C_DIS
LIN {X -12.1687,Y -26.6657,Z 61,A -120.1895,B 24.8452,C -2.8706,E1 24.9367,E2 -516.9516} C_DIS
LIN {X -9.8831,Y -27.5959,Z 61,A -115.7886,B 24.8461,C -2.8624,E1 24.9482,E2 -521.3421} C_DIS
LIN {X -7.5745,Y -28.3163,Z 61,A -110.1643,B 24.8455,C -2.8677,E1 24.9633,E2 -526.9882} C_DIS
LIN {X -5.3996,Y -28.8105,Z 61,A -106.7815,B 24.8467,C -2.8565,E1 24.9725,E2 -530.3484} C_DIS
LIN {X -3.2183,Y -29.1348,Z 61,A -101.43,B 24.8457,C -2.866,E1 24.9874,E2 -535.7263} C_DIS
LIN {X -0.874,Y -29.2987,Z 61,A -97.6216,B 24.8465,C -2.8584,E1 24.998,E2 -539.5177} C_DIS
LIN {X -0.874,Y -29.2987,Z 61,A -97.6216,B 24.8465,C -2.8584,E1 24.998,E2 -539.5177} C_DIS
Enddeposition()
LIN {X 0.1546,Y -28.3231,Z 61,A -97.1654,B 24.8463,C -2.8606,E1 24.9992,E2 -539.9789} C_DIS
Startdeposition()
$VEL.CP = VEL_PRINT
LIN {X -1.6281,Y -28.2793,Z 61,A -100.6801,B 24.8463,C -2.861,E1 24.9894,E2 -536.4647} C_DIS
LIN {X -3.5115,Y -28.1079,Z 61,A -105.5094,B 24.8472,C -2.8522,E1 24.976,E2 -531.6114} C_DIS
LIN {X -6.0246,Y -27.6786,Z 61,A -109.8184,B 24.8461,C -2.8617,E1 24.9642,E2 -527.3202} C_DIS
LIN {X -7.7596,Y -27.2433,Z 61,A -114.1434,B 24.8466,C -2.8577,E1 24.9525,E2 -522.9792} C_DIS
LIN {X -9.9253,Y -26.5312,Z 61,A -117.7716,B 24.8453,C -2.8698,E1 24.943,E2 -519.3728} C_DIS
LIN {X -11.3516,Y -25.9528,Z 61,A -121.4847,B 24.8455,C -2.8679,E1 24.9334,E2 -515.6467} C_DIS
LIN {X -13.1656,Y -25.0813,Z 61,A -125.5479,B 24.8449,C -2.8729,E1 24.9233,E2 -511.5844} C_DIS
LIN {X -14.5759,Y -24.2887,Z 61,A -128.8593,B 24.8445,C -2.8771,E1 24.9153,E2 -508.2732} C_DIS
LIN {X -15.8246,Y -23.4945,Z 61,A -131.8972,B 24.844,C -2.8813,E1 24.9082,E2 -505.2355} C_DIS
LIN {X -17.3843,Y -22.3646,Z 61,A -135.4697,B 24.843,C -2.8904,E1 24.9003,E2 -501.6718} C_DIS
LIN {X -18.6204,Y -21.3468,Z 61,A -138.7137,B 24.8424,C -2.8963,E1 24.8933,E2 -498.4295} C_DIS
LIN {X -20.0264,Y -20.0344,Z 61,A -143.168,B 24.842,C -2.9001,E1 24.8844,E2 -493.9656} C_DIS
LIN {X -21.1323,Y -18.8635,Z 61,A -146.9504,B 24.8416,C -2.9035,E1 24.8773,E2 -490.1745} C_DIS
LIN {X -22.8644,Y -16.722,Z 61,A -151.549,B 24.8394,C -2.9232,E1 24.8695,E2 -485.6011} C_DIS
LIN {X -23.7088,Y -15.5018,Z 61,A -154.4545,B 24.8385,C -2.9312,E1 24.865,E2 -482.7004} C_DIS
LIN {X -24.5221,Y -14.1799,Z 61,A -158.1624,B 24.8381,C -2.9355,E1 24.8597,E2 -478.9836} C_DIS
LIN {X -25.5701,Y -12.1888,Z 61,A -163.0791,B 24.837,C -2.9455,E1 24.8536,E2 -474.0642} C_DIS
LIN {X -26.7139,Y -9.422,Z 61,A -168.5538,B 24.8346,C -2.9663,E1 24.8481,E2 -468.6087} C_DIS
LIN {X -27.3935,Y -7.213,Z 61,A -173.4105,B 24.8332,C -2.9789,E1 24.8443,E2 -463.754} C_DIS
LIN {X -27.785,Y -5.5157,Z 61,A -177.1937,B 24.8322,C -2.9879,E1 24.8422,E2 -459.97} C_DIS
LIN {X -28.1427,Y -3.2238,Z 61,A 178.3701,B 24.8304,C -3.0038,E1 24.8405,E2 -455.5456} C_DIS
LIN {X -28.3168,Y -0.7428,Z 61,A 172.4953,B 24.8292,C -3.0144,E1 24.8398,E2 -449.6607} C_DIS
LIN {X -28.2899,Y 1.4495,Z 61,A 169.0109,B 24.827,C -3.0339,E1 24.8401,E2 -446.2021} C_DIS
LIN {X -28.1403,Y 3.245,Z 61,A 165.2171,B 24.8258,C -3.0444,E1 24.8412,E2 -442.4106} C_DIS
LIN {X -27.8585,Y 5.1304,Z 61,A 161.3619,B 24.8244,C -3.0564,E1 24.8429,E2 -438.5612} C_DIS
LIN {X -27.4136,Y 7.1349,Z 61,A 157.0875,B 24.823,C -3.0684,E1 24.8457,E2 -434.2907} C_DIS
LIN {X -26.8624,Y 8.99,Z 61,A 153.271,B 24.8216,C -3.0809,E1 24.8489,E2 -430.4822} C_DIS
LIN {X -26.2813,Y 10.5695,Z 61,A 149.9634,B 24.8203,C -3.0916,E1 24.8522,E2 -427.1817} C_DIS
LIN {X -25.688,Y 11.9387,Z 61,A 146.9675,B 24.8193,C -3.1006,E1 24.8556,E2 -424.1908} C_DIS
LIN {X -25.1078,Y 13.1153,Z 61,A 144.0124,B 24.8186,C -3.1063,E1 24.8594,E2 -421.2336} C_DIS
LIN {X -24.4084,Y 14.3748,Z 61,A 141.19,B 24.8176,C -3.1151,E1 24.8633,E2 -418.4174} C_DIS
LIN {X -23.484,Y 15.84,Z 61,A 137.506,B 24.8166,C -3.1234,E1 24.869,E2 -414.735} C_DIS
LIN {X -22.1479,Y 17.6604,Z 61,A 133.3121,B 24.8149,C -3.1377,E1 24.876,E2 -410.5553} C_DIS
LIN {X -21.1426,Y 18.8521,Z 61,A 129.6276,B 24.8144,C -3.142,E1 24.8828,E2 -406.8644} C_DIS
LIN {X -19.6224,Y 20.4296,Z 61,A 125.3989,B 24.813,C -3.1538,E1 24.8911,E2 -402.6459} C_DIS
LIN {X -18.2028,Y 21.7038,Z 61,A 121.3568,B 24.8121,C -3.161,E1 24.8997,E2 -398.6051} C_DIS
LIN {X -16.5654,Y 22.9785,Z 61,A 117.2768,B 24.811,C -3.1703,E1 24.9087,E2 -394.5329} C_DIS
LIN {X -14.6403,Y 24.2502,Z 61,A 112.6162,B 24.81,C -3.1789,E1 24.9197,E2 -389.8779} C_DIS
LIN {X -13.2683,Y 25.0272,Z 61,A 109.7488,B 24.809,C -3.1866,E1 24.9267,E2 -387.0208} C_DIS
LIN {X -12.1489,Y 25.5893,Z 61,A 106.9211,B 24.8088,C -3.1883,E1 24.9338,E2 -384.1898} C_DIS
LIN {X -10.5567,Y 26.2864,Z 61,A 103.2286,B 24.8084,C -3.1918,E1 24.9433,E2 -380.4971} C_DIS
LIN {X -8.5042,Y 27.0199,Z 61,A 99.1858,B 24.8074,C -3.1999,E1 24.954,E2 -376.4662} C_DIS
LIN {X -7.1078,Y 27.4206,Z 61,A 96.0872,B 24.8072,C -3.2016,E1 24.9623,E2 -373.3667} C_DIS
LIN {X -5.4764,Y 27.7925,Z 61,A 92.6862,B 24.8069,C -3.2042,E1 24.9716,E2 -369.968} C_DIS
LIN {X -3.7034,Y 28.0836,Z 61,A 88.89,B 24.8068,C -3.2052,E1 24.9821,E2 -366.171} C_DIS
LIN {X -2.0539,Y 28.2526,Z 61,A 85.7289,B 24.8064,C -3.2084,E1 24.9909,E2 -363.016} C_DIS
LIN {X -0.7638,Y 28.3163,Z 61,A 82.9401,B 24.8064,C -3.2077,E1 24.9987,E2 -360.2249} C_DIS
LIN {X 1.2689,Y 28.2984,Z 61,A 78.9457,B 24.8064,C -3.2092,E1 25.0098,E2 -356.2349} C_DIS
LIN {X 3.8634,Y 28.0618,Z 61,A 72.4754,B 24.8078,C -3.1972,E1 25.0278,E2 -349.7408} C_DIS
LIN {X 6.4688,Y 27.5784,Z 61,A 68.2365,B 24.8068,C -3.2054,E1 25.0393,E2 -345.5269} C_DIS
LIN {X 8.4813,Y 27.0274,Z 61,A 63.8911,B 24.8073,C -3.2013,E1 25.051,E2 -341.1791} C_DIS
LIN {X 10.2404,Y 26.4112,Z 61,A 60.3892,B 24.8073,C -3.2006,E1 25.0601,E2 -337.683} C_DIS
LIN {X 11.724,Y 25.7864,Z 61,A 56.6677,B 24.8083,C -3.1923,E1 25.0697,E2 -333.9509} C_DIS
LIN {X 13.3246,Y 24.9976,Z 61,A 53.5482,B 24.8083,C -3.1929,E1 25.0774,E2 -330.8414} C_DIS
LIN {X 14.5742,Y 24.2904,Z 61,A 50.4034,B 24.8091,C -3.1862,E1 25.085,E2 -327.6903} C_DIS
LIN {X 16.3891,Y 23.1043,Z 61,A 46.2294,B 24.8096,C -3.1816,E1 25.0946,E2 -323.5193} C_DIS
LIN {X 17.8699,Y 21.9789,Z 61,A 42.0169,B 24.811,C -3.1699,E1 25.1038,E2 -319.2949} C_DIS
LIN {X 19.5625,Y 20.4874,Z 61,A 37.6343,B 24.8119,C -3.163,E1 25.1128,E2 -314.9135} C_DIS
LIN {X 21.1645,Y 18.8274,Z 61,A 33.4849,B 24.8124,C -3.1588,E1 25.1207,E2 -310.7725} C_DIS
LIN {X 22.3824,Y 17.3621,Z 61,A 29.0484,B 24.8142,C -3.1432,E1 25.1285,E2 -306.3196} C_DIS
LIN {X 23.7453,Y 15.4465,Z 61,A 23.7198,B 24.8164,C -3.1248,E1 25.1368,E2 -300.9737} C_DIS
LIN {X 25.5941,Y 12.1395,Z 61,A 16.0439,B 24.8188,C -3.1041,E1 25.1467,E2 -293.2896} C_DIS
LIN {X 26.9677,Y 8.669,Z 61,A 9.9488,B 24.8193,C -3.1002,E1 25.1526,E2 -287.2191} C_DIS
LIN {X 27.2764,Y 7.6427,Z 61,A 6.7761,B 24.8215,C -3.0815,E1 25.155,E2 -284.0204} C_DIS
LIN {X 27.9416,Y 4.6549,Z 61,A 1.448,B 24.8224,C -3.0734,E1 25.1579,E2 -278.7042} C_DIS
LIN {X 28.1416,Y 3.2341,Z 61,A -2.2331,B 24.8246,C -3.0549,E1 25.1592,E2 -275.001} C_DIS
LIN {X 28.3255,Y 0.062,Z 61,A -7.7196,B 24.8255,C -3.0466,E1 25.1598,E2 -269.5274} C_DIS
LIN {X 28.2794,Y -1.6345,Z 61,A -11.5215,B 24.8273,C -3.0312,E1 25.1593,E2 -265.7118} C_DIS
LIN {X 28.0986,Y -3.5883,Z 61,A -15.3256,B 24.8285,C -3.0209,E1 25.1582,E2 -261.9056} C_DIS
LIN {X 27.8037,Y -5.4161,Z 61,A -18.6931,B 24.8293,C -3.0139,E1 25.1566,E2 -258.5414} C_DIS
LIN {X 27.5563,Y -6.5624,Z 61,A -21.5615,B 24.8308,C -3.0004,E1 25.1548,E2 -255.6576} C_DIS
LIN {X 26.9726,Y -8.6539,Z 61,A -25.8879,B 24.8322,C -2.9878,E1 25.1513,E2 -251.326} C_DIS
LIN {X 26.1618,Y -10.8601,Z 61,A -31.1669,B 24.8345,C -2.9672,E1 25.1459,E2 -246.0274} C_DIS
LIN {X 25.2011,Y -12.9348,Z 61,A -35.4357,B 24.8356,C -2.9581,E1 25.1406,E2 -241.7599} C_DIS
LIN {X 24.0955,Y -14.894,Z 61,A -39.6367,B 24.8365,C -2.9496,E1 25.1347,E2 -237.5603} C_DIS
LIN {X 23.0793,Y -16.4241,Z 61,A -43.213,B 24.8374,C -2.9412,E1 25.129,E2 -233.9819} C_DIS
LIN {X 22.1093,Y -17.7077,Z 61,A -46.4413,B 24.8383,C -2.933,E1 25.1235,E2 -230.7495} C_DIS
LIN {X 21.0518,Y -18.9535,Z 61,A -49.6776,B 24.8392,C -2.9256,E1 25.1175,E2 -227.5101} C_DIS
LIN {X 20.0299,Y -20.0306,Z 61,A -52.9201,B 24.8403,C -2.9156,E1 25.1112,E2 -224.2577} C_DIS
LIN {X 18.5784,Y -21.3834,Z 61,A -56.6637,B 24.8409,C -2.9096,E1 25.1034,E2 -220.5151} C_DIS
LIN {X 17.4008,Y -22.3525,Z 61,A -59.9055,B 24.8418,C -2.9013,E1 25.0964,E2 -217.2656} C_DIS
LIN {X 15.9265,Y -23.4254,Z 61,A -63.2898,B 24.8423,C -2.8974,E1 25.0886,E2 -213.8838} C_DIS
LIN {X 14.8733,Y -24.1082,Z 61,A -66.5542,B 24.8437,C -2.8846,E1 25.0809,E2 -210.5994} C_DIS
LIN {X 12.4588,Y -25.4389,Z 61,A -71.2372,B 24.8436,C -2.8852,E1 25.0694,E2 -205.9311} C_DIS
LIN {X 10.9407,Y -26.1287,Z 61,A -74.4076,B 24.8439,C -2.8824,E1 25.0613,E2 -202.7618} C_DIS
LIN {X 9.41,Y -26.7181,Z 61,A -78.8577,B 24.8457,C -2.866,E1 25.0495,E2 -198.2823} C_DIS
LIN {X 6.6737,Y -27.5294,Z 61,A -84.4753,B 24.8461,C -2.8617,E1 25.0344,E2 -192.6633} C_DIS
LIN {X 4.915,Y -27.8973,Z 61,A -88.2946,B 24.8467,C -2.8569,E1 25.0239,E2 -188.8371} C_DIS
LIN {X 2.2093,Y -28.2405,Z 61,A -93.2001,B 24.8463,C -2.8599,E1 25.0103,E2 -183.9418} C_DIS
LIN {X 0.3389,Y -28.3244,Z 61,A -97.1572,B 24.8466,C -2.8571,E1 24.9992,E2 -179.9789} C_DIS
LIN {X 0.3389,Y -28.3244,Z 61,A -97.1572,B 24.8466,C -2.8571,E1 24.9992,E2 -179.9789} C_DIS
Enddeposition()
LIN {X 0.1616,Y -27.3391,Z 61,A -97.2293,B 24.8445,C -2.877,E1 24.9992,E2 -179.9542} C_DIS
Startdeposition()
$VEL.CP = VEL_PRINT
LIN {X 1.5856,Y -27.2954,Z 61,A -92.7403,B 24.8428,C -2.8921,E1 25.0118,E2 -184.4782} C_DIS
LIN {X 3.3737,Y -27.1329,Z 61,A -88.6453,B 24.8422,C -2.8975,E1 25.0232,E2 -188.5832} C_DIS
LIN {X 5.3468,Y -26.8142,Z 61,A -83.9538,B 24.8413,C -2.906,E1 25.0361,E2 -193.2894} C_DIS
LIN {X 7.9347,Y -26.1656,Z 61,A -78.9842,B 24.8413,C -2.9054,E1 25.0494,E2 -198.2495} C_DIS
LIN {X 9.9561,Y -25.4646,Z 61,A -74.8527,B 24.8412,C -2.9074,E1 25.0603,E2 -202.3772} C_DIS
LIN {X 11.5163,Y -24.7981,Z 61,A -70.379,B 24.8395,C -2.9226,E1 25.0717,E2 -206.876} C_DIS
LIN {X 14.4805,Y -23.1924,Z 61,A -63.9823,B 24.8389,C -2.9276,E1 25.0872,E2 -213.2652} C_DIS
LIN {X 16.0456,Y -22.1385,Z 61,A -60.1617,B 24.8383,C -2.9338,E1 25.096,E2 -217.0876} C_DIS
LIN {X 17.5113,Y -20.9983,Z 61,A -55.9548,B 24.8369,C -2.9458,E1 25.1051,E2 -221.3069} C_DIS
LIN {X 18.8465,Y -19.8092,Z 61,A -52.1827,B 24.8359,C -2.9546,E1 25.1128,E2 -225.0846} C_DIS
LIN {X 20.3664,Y -18.2422,Z 61,A -47.731,B 24.8349,C -2.9644,E1 25.1213,E2 -229.5399} C_DIS
LIN {X 21.9013,Y -16.3679,Z 61,A -42.9465,B 24.8338,C -2.974,E1 25.1296,E2 -234.3249} C_DIS
LIN {X 22.9213,Y -14.9062,Z 61,A -39.1937,B 24.8326,C -2.9844,E1 25.1355,E2 -238.0836} C_DIS
LIN {X 23.7311,Y -13.5796,Z 61,A -36.0792,B 24.8318,C -2.9918,E1 25.1399,E2 -241.1996} C_DIS
LIN {X 24.4877,Y -12.1624,Z 61,A -33.0953,B 24.8312,C -2.9968,E1 25.1437,E2 -244.1797} C_DIS
LIN {X 25.2146,Y -10.5716,Z 61,A -29.0796,B 24.8295,C -3.0119,E1 25.1483,E2 -248.2092} C_DIS
LIN {X 25.935,Y -8.6574,Z 61,A -24.2105,B 24.8272,C -3.032,E1 25.1528,E2 -253.0986} C_DIS
LIN {X 26.4815,Y -6.8043,Z 61,A -19.8049,B 24.8253,C -3.0489,E1 25.156,E2 -257.5188} C_DIS
LIN {X 27.081,Y -3.7675,Z 61,A -14.1111,B 24.8241,C -3.0592,E1 25.1586,E2 -263.2036} C_DIS
LIN {X 27.2969,Y -1.5618,Z 61,A -9.9099,B 24.823,C -3.0682,E1 25.1596,E2 -267.4013} C_DIS
LIN {X 27.3398,Y -0.281,Z 61,A -5.9764,B 24.8202,C -3.0921,E1 25.1597,E2 -271.368} C_DIS
LIN {X 27.1225,Y 3.4555,Z 61,A 0.2901,B 24.8197,C -3.0969,E1 25.1584,E2 -277.6086} C_DIS
LIN {X 26.721,Y 5.7929,Z 61,A 7.0539,B 24.8153,C -3.1339,E1 25.1547,E2 -284.4208} C_DIS
LIN {X 25.5262,Y 9.7975,Z 61,A 15.4449,B 24.8129,C -3.1547,E1 25.1472,E2 -292.8136} C_DIS
LIN {X 24.4822,Y 12.1734,Z 61,A 20.3908,B 24.8118,C -3.1636,E1 25.1413,E2 -297.7539} C_DIS
LIN {X 23.0576,Y 14.6944,Z 61,A 25.7229,B 24.811,C -3.1705,E1 25.1337,E2 -303.0752} C_DIS
LIN {X 22.0793,Y 16.1268,Z 61,A 29.6402,B 24.8095,C -3.1826,E1 25.1274,E2 -307.0021} C_DIS
LIN {X 20.9042,Y 17.624,Z 61,A 33.2442,B 24.8089,C -3.1874,E1 25.1211,E2 -310.6006} C_DIS
LIN {X 20.0254,Y 18.616,Z 61,A 36.3044,B 24.8078,C -3.1966,E1 25.1153,E2 -313.6692} C_DIS
LIN {X 18.4496,Y 20.1788,Z 61,A 40.3479,B 24.8075,C -3.1993,E1 25.1072,E2 -317.7021} C_DIS
LIN {X 17.4016,Y 21.0894,Z 61,A 43.5784,B 24.8064,C -3.2082,E1 25.1003,E2 -320.9413} C_DIS
LIN {X 16.2487,Y 21.9901,Z 61,A 46.6654,B 24.8058,C -3.2138,E1 25.0934,E2 -324.0303} C_DIS
LIN {X 15.0141,Y 22.8506,Z 61,A 49.8765,B 24.8051,C -3.2194,E1 25.086,E2 -327.2439} C_DIS
LIN {X 13.562,Y 23.7413,Z 61,A 53.7371,B 24.8041,C -3.2275,E1 25.0767,E2 -331.112} C_DIS
LIN {X 12.1043,Y 24.5165,Z 61,A 57.0968,B 24.8037,C -3.2308,E1 25.0683,E2 -334.4702} C_DIS
LIN {X 10.5328,Y 25.2317,Z 61,A 60.3953,B 24.8037,C -3.2314,E1 25.0599,E2 -337.7622} C_DIS
LIN {X 9.3055,Y 25.7096,Z 61,A 63.0884,B 24.8034,C -3.2332,E1 25.0529,E2 -340.4539} C_DIS
LIN {X 7.8306,Y 26.1961,Z 61,A 66.8952,B 24.8024,C -3.2411,E1 25.0427,E2 -344.2726} C_DIS
LIN {X 5.7553,Y 26.7292,Z 61,A 71.2157,B 24.8024,C -3.2418,E1 25.031,E2 -348.5886} C_DIS
LIN {X 3.3155,Y 27.1395,Z 61,A 76.333,B 24.8022,C -3.2426,E1 25.0168,E2 -353.7031} C_DIS
LIN {X 1.505,Y 27.3002,Z 61,A 80.3967,B 24.8019,C -3.245,E1 25.0055,E2 -357.7706} C_DIS
LIN {X -0.8423,Y 27.3287,Z 61,A 85.1547,B 24.8023,C -3.2424,E1 24.9923,E2 -362.5228} C_DIS
LIN {X -2.6938,Y 27.2091,Z 61,A 89.0307,B 24.8025,C -3.2406,E1 24.9815,E2 -366.396} C_DIS
LIN {X -4.9115,Y 26.8964,Z 61,A 93.401,B 24.8032,C -3.2347,E1 24.9695,E2 -370.7563} C_DIS
LIN {X -6.3361,Y 26.5976,Z 61,A 97.0803,B 24.8029,C -3.2372,E1 24.9594,E2 -374.4462} C_DIS
LIN {X -8.7049,Y 25.919,Z 61,A 101.7273,B 24.8041,C -3.2273,E1 24.9471,E2 -379.0778} C_DIS
LIN {X -10.2443,Y 25.3501,Z 61,A 105.0406,B 24.8048,C -3.2219,E1 24.9384,E2 -382.3851} C_DIS
LIN {X -11.4401,Y 24.8333,Z 61,A 107.9636,B 24.8051,C -3.2194,E1 24.931,E2 -385.3093} C_DIS
LIN {X -12.9574,Y 24.0766,Z 61,A 111.5981,B 24.8057,C -3.2143,E1 24.922,E2 -388.9414} C_DIS
LIN {X -14.4236,Y 23.2279,Z 61,A 115.0686,B 24.8065,C -3.2074,E1 24.9137,E2 -392.4062} C_DIS
LIN {X -15.8856,Y 22.2535,Z 61,A 118.6982,B 24.8074,C -3.2,E1 24.9053,E2 -396.0302} C_DIS
LIN {X -17.0622,Y 21.365,Z 61,A 121.56,B 24.8084,C -3.192,E1 24.899,E2 -398.8834} C_DIS
LIN {X -17.98,Y 20.5983,Z 61,A 124.7985,B 24.8084,C -3.1916,E1 24.8922,E2 -402.1336} C_DIS
LIN {X -19.731,Y 18.9278,Z 61,A 129.9981,B 24.8098,C -3.1806,E1 24.8819,E2 -407.3289} C_DIS
LIN {X -21.1264,Y 17.3568,Z 61,A 133.9011,B 24.8115,C -3.1663,E1 24.8749,E2 -411.2154} C_DIS
LIN {X -22.1038,Y 16.0929,Z 61,A 137.0081,B 24.8127,C -3.156,E1 24.8697,E2 -414.3127} C_DIS
LIN {X -22.7675,Y 15.1401,Z 61,A 139.6158,B 24.8134,C -3.1506,E1 24.8656,E2 -416.9203} C_DIS
LIN {X -23.6248,Y 13.7646,Z 61,A 143.3346,B 24.8142,C -3.1432,E1 24.8602,E2 -420.6405} C_DIS
LIN {X -24.4285,Y 12.2818,Z 61,A 146.9001,B 24.8154,C -3.1333,E1 24.8556,E2 -424.2014} C_DIS
LIN {X -25.2272,Y 10.5425,Z 61,A 150.4437,B 24.8171,C -3.1187,E1 24.8516,E2 -427.7295} C_DIS
LIN {X -25.6234,Y 9.5412,Z 61,A 152.937,B 24.8178,C -3.1134,E1 24.8492,E2 -430.2241} C_DIS
LIN {X -26.048,Y 8.3098,Z 61,A 156.4172,B 24.8182,C -3.1097,E1 24.8462,E2 -433.7154} C_DIS
LIN {X -26.808,Y 5.3776,Z 61,A 163.0799,B 24.8203,C -3.0921,E1 24.842,E2 -440.3749} C_DIS
LIN {X -27.2276,Y 2.4951,Z 61,A 168.082,B 24.8232,C -3.0664,E1 24.8403,E2 -445.3453} C_DIS
LIN {X -27.3122,Y 1.275,Z 61,A 170.7083,B 24.8241,C -3.0587,E1 24.8399,E2 -447.9692} C_DIS
LIN {X -27.3279,Y -0.8603,Z 61,A 175.7265,B 24.8254,C -3.0481,E1 24.8399,E2 -452.9921} C_DIS
LIN {X -27.2,Y -2.7795,Z 61,A 179.5726,B 24.8269,C -3.0345,E1 24.8409,E2 -456.8287} C_DIS
LIN {X -26.9388,Y -4.6796,Z 61,A -176.2938,B 24.8282,C -3.0229,E1 24.8427,E2 -460.9593} C_DIS
LIN {X -26.527,Y -6.6263,Z 61,A -172.0698,B 24.8296,C -3.0108,E1 24.8453,E2 -465.179} C_DIS
LIN {X -25.9376,Y -8.6497,Z 61,A -167.1745,B 24.8307,C -3.001,E1 24.8494,E2 -470.0789} C_DIS
LIN {X -24.895,Y -11.3037,Z 61,A -162.3086,B 24.8334,C -2.9772,E1 24.8546,E2 -474.9149} C_DIS
LIN {X -24.2929,Y -12.5474,Z 61,A -158.2468,B 24.8334,C -2.9769,E1 24.8597,E2 -478.9979} C_DIS
LIN {X -23.0247,Y -14.7456,Z 61,A -153.6128,B 24.8355,C -2.9588,E1 24.8664,E2 -483.6123} C_DIS
LIN {X -22.031,Y -16.1928,Z 61,A -150.0825,B 24.8366,C -2.9489,E1 24.872,E2 -487.1362} C_DIS
LIN {X -21.3567,Y -17.0729,Z 61,A -147.6245,B 24.8371,C -2.9444,E1 24.8763,E2 -489.5951} C_DIS
LIN {X -20.4312,Y -18.1699,Z 61,A -144.7378,B 24.8379,C -2.9369,E1 24.8815,E2 -492.4769} C_DIS
LIN {X -19.2022,Y -19.464,Z 61,A -140.9843,B 24.8388,C -2.9292,E1 24.8888,E2 -496.2282} C_DIS
LIN {X -18.3477,Y -20.272,Z 61,A -138.4544,B 24.8392,C -2.9248,E1 24.894,E2 -498.758} C_DIS
LIN {X -17.1627,Y -21.2842,Z 61,A -134.5565,B 24.8394,C -2.9236,E1 24.9024,E2 -502.6677} C_DIS
LIN {X -15.1176,Y -22.7823,Z 61,A -129.5805,B 24.8406,C -2.9124,E1 24.9138,E2 -507.6341} C_DIS
LIN {X -12.8442,Y -24.1363,Z 61,A -123.6028,B 24.8411,C -2.9084,E1 24.9283,E2 -513.6197} C_DIS
LIN {X -10.821,Y -25.1085,Z 61,A -118.9053,B 24.8416,C -2.9032,E1 24.9402,E2 -518.3164} C_DIS
LIN {X -8.7705,Y -25.8969,Z 61,A -114.534,B 24.8423,C -2.8974,E1 24.9517,E2 -522.6825} C_DIS
LIN {X -6.4043,Y -26.5812,Z 61,A -109.1496,B 24.8423,C -2.8963,E1 24.9662,E2 -528.0724} C_DIS
LIN {X -4.4421,Y -26.9785,Z 61,A -104.4429,B 24.842,C -2.8995,E1 24.9792,E2 -532.7916} C_DIS
LIN {X -0.9432,Y -27.3257,Z 61,A -98.5982,B 24.8436,C -2.8852,E1 24.9954,E2 -538.6048} C_DIS
LIN {X -0.9432,Y -27.3257,Z 61,A -98.5982,B 24.8436,C -2.8852,E1 24.9954,E2 -538.6048} C_DIS
Enddeposition()
LIN {X 0.1612,Y -26.3525,Z 61,A -96.8431,B 24.8422,C -2.8976,E1 25.0004,E2 -540.3895} C_DIS
Startdeposition()
$VEL.CP = VEL_PRINT
LIN {X -1.1365,Y -26.3322,Z 61,A -100.9068,B 24.8435,C -2.8864,E1 24.989,E2 -536.2982} C_DIS
LIN {X -3.7756,Y -26.0847,Z 61,A -105.944,B 24.8427,C -2.8933,E1 24.975,E2 -531.2742} C_DIS
LIN {X -5.4318,Y -25.7913,Z 61,A -110.0572,B 24.843,C -2.8909,E1 24.9637,E2 -527.1508} C_DIS
LIN {X -7.543,Y -25.2543,Z 61,A -114.5628,B 24.8425,C -2.8956,E1 24.9516,E2 -522.6495} C_DIS
LIN {X -9.417,Y -24.6171,Z 61,A -118.3364,B 24.8416,C -2.9033,E1 24.9417,E2 -518.8868} C_DIS
LIN {X -10.7549,Y -24.0622,Z 61,A -121.7104,B 24.8414,C -2.9048,E1 24.9331,E2 -515.5085} C_DIS
LIN {X -12.2947,Y -23.3135,Z 61,A -126.2389,B 24.8416,C -2.9034,E1 24.9218,E2 -510.9644} C_DIS
LIN {X -14.4097,Y -22.0692,Z 61,A -131.8039,B 24.8409,C -2.9096,E1 24.9086,E2 -505.3967} C_DIS
LIN {X -16.939,Y -20.1931,Z 61,A -137.8173,B 24.839,C -2.9272,E1 24.8954,E2 -499.4032} C_DIS
LIN {X -18.0356,Y -19.2196,Z 61,A -140.8165,B 24.8382,C -2.9347,E1 24.8892,E2 -496.4097} C_DIS
LIN {X -19.2206,Y -18.0346,Z 61,A -144.5924,B 24.8374,C -2.9414,E1 24.8818,E2 -492.6336} C_DIS
LIN {X -20.1207,Y -17.0243,Z 61,A -147.2505,B 24.8365,C -2.9497,E1 24.877,E2 -489.9835} C_DIS
LIN {X -21.0879,Y -15.8106,Z 61,A -151.6595,B 24.8363,C -2.9511,E1 24.8694,E2 -485.557} C_DIS
LIN {X -22.7598,Y -13.2924,Z 61,A -158.4814,B 24.8346,C -2.9663,E1 24.8594,E2 -478.7365} C_DIS
LIN {X -23.7415,Y -11.4463,Z 61,A -163.2645,B 24.8334,C -2.9772,E1 24.8535,E2 -473.9537} C_DIS
LIN {X -25.1178,Y -7.9868,Z 61,A -170.6288,B 24.8303,C -3.0044,E1 24.8464,E2 -466.6131} C_DIS
LIN {X -25.6483,Y -6.0713,Z 61,A -174.9185,B 24.8289,C -3.0174,E1 24.8434,E2 -462.3294} C_DIS
LIN {X -26.0341,Y -4.1121,Z 61,A -178.5053,B 24.8269,C -3.0347,E1 24.8416,E2 -458.7629} C_DIS
LIN {X -26.2219,Y -2.6562,Z 61,A 177.654,B 24.8262,C -3.0409,E1 24.8404,E2 -454.9141} C_DIS
LIN {X -26.3383,Y -0.9692,Z 61,A 173.4302,B 24.8252,C -3.0494,E1 24.8398,E2 -450.6851} C_DIS
LIN {X -26.3337,Y 1.1004,Z 61,A 169.3466,B 24.8233,C -3.0656,E1 24.8401,E2 -446.6158} C_DIS
LIN {X -26.2175,Y 2.7058,Z 61,A 166.0553,B 24.8219,C -3.0777,E1 24.8409,E2 -443.3336} C_DIS
LIN {X -26.0325,Y 4.1216,Z 61,A 162.6181,B 24.821,C -3.0856,E1 24.8422,E2 -439.8948} C_DIS
LIN {X -25.6846,Y 5.914,Z 61,A 158.8579,B 24.8194,C -3.099,E1 24.8444,E2 -436.1445} C_DIS
LIN {X -25.2561,Y 7.537,Z 61,A 154.9073,B 24.8183,C -3.1085,E1 24.8474,E2 -432.1938} C_DIS
LIN {X -24.6955,Y 9.2101,Z 61,A 151.4435,B 24.8167,C -3.122,E1 24.8506,E2 -428.7429} C_DIS
LIN {X -24.0155,Y 10.8597,Z 61,A 146.777,B 24.8159,C -3.1291,E1 24.8558,E2 -424.0675} C_DIS
LIN {X -22.9328,Y 12.9913,Z 61,A 142.109,B 24.8138,C -3.1468,E1 24.8619,E2 -419.4172} C_DIS
LIN {X -21.9018,Y 14.663,Z 61,A 136.9725,B 24.813,C -3.1535,E1 24.8697,E2 -414.2708} C_DIS
LIN {X -20.2306,Y 16.8939,Z 61,A 131.9234,B 24.8104,C -3.175,E1 24.8784,E2 -409.2494} C_DIS
LIN {X -19.0773,Y 18.1866,Z 61,A 127.6738,B 24.8097,C -3.1812,E1 24.8864,E2 -404.9959} C_DIS
LIN {X -17.8039,Y 19.4345,Z 61,A 123.995,B 24.8085,C -3.1913,E1 24.8938,E2 -401.3261} C_DIS
LIN {X -16.3281,Y 20.6899,Z 61,A 119.2747,B 24.8078,C -3.197,E1 24.9041,E2 -396.6016} C_DIS
LIN {X -14.9753,Y 21.6891,Z 61,A 115.7533,B 24.8068,C -3.205,E1 24.9121,E2 -393.0873} C_DIS
LIN {X -13.0558,Y 22.8961,Z 61,A 111.549,B 24.8052,C -3.2187,E1 24.9221,E2 -388.9026} C_DIS
LIN {X -11.6711,Y 23.6318,Z 61,A 107.5166,B 24.805,C -3.2198,E1 24.9321,E2 -384.862} C_DIS
LIN {X -9.9318,Y 24.4138,Z 61,A 103.8456,B 24.8039,C -3.229,E1 24.9415,E2 -381.2044} C_DIS
LIN {X -8.9079,Y 24.8055,Z 61,A 100.6514,B 24.8043,C -3.2261,E1 24.9499,E2 -377.9969} C_DIS
LIN {X -6.0782,Y 25.6466,Z 61,A 94.3314,B 24.8034,C -3.2333,E1 24.9669,E2 -371.6842} C_DIS
LIN {X -3.8629,Y 26.0726,Z 61,A 89.6576,B 24.8027,C -3.2385,E1 24.9798,E2 -367.0186} C_DIS
LIN {X -1.8876,Y 26.2893,Z 61,A 85.3044,B 24.8025,C -3.2403,E1 24.9918,E2 -362.6674} C_DIS
LIN {X -0.2218,Y 26.3558,Z 61,A 81.6986,B 24.8024,C -3.2414,E1 25.0019,E2 -359.0638} C_DIS
LIN {X 1.8771,Y 26.29,Z 61,A 77.5201,B 24.802,C -3.2449,E1 25.0135,E2 -354.8951} C_DIS
LIN {X 3.5705,Y 26.1141,Z 61,A 73.4258,B 24.8025,C -3.2408,E1 25.0249,E2 -350.7941} C_DIS
LIN {X 5.4668,Y 25.784,Z 61,A 69.2579,B 24.8026,C -3.2393,E1 25.0363,E2 -346.6274} C_DIS
LIN {X 6.8843,Y 25.4417,Z 61,A 66.1736,B 24.8028,C -3.2382,E1 25.0447,E2 -343.5452} C_DIS
LIN {X 8.4232,Y 24.9745,Z 61,A 62.4495,B 24.8034,C -3.2333,E1 25.0546,E2 -339.8166} C_DIS
LIN {X 10.8143,Y 24.036,Z 61,A 57.0944,B 24.8038,C -3.2299,E1 25.0684,E2 -334.4656} C_DIS
LIN {X 11.8708,Y 23.5325,Z 61,A 54.0666,B 24.8047,C -3.222,E1 25.0759,E2 -331.4275} C_DIS
LIN {X 14.1526,Y 22.2348,Z 61,A 48.8363,B 24.8052,C -3.2186,E1 25.0884,E2 -326.2052} C_DIS
LIN {X 15.5107,Y 21.3096,Z 61,A 45.5603,B 24.8055,C -3.2158,E1 25.0959,E2 -322.9338} C_DIS
LIN {X 16.9322,Y 20.1987,Z 61,A 41.3014,B 24.8068,C -3.2052,E1 25.1052,E2 -318.6659} C_DIS
LIN {X 18.9008,Y 18.3697,Z 61,A 36.1323,B 24.8074,C -3.2006,E1 25.1156,E2 -313.5072} C_DIS
LIN {X 19.73,Y 17.4759,Z 61,A 33.1952,B 24.8084,C -3.1917,E1 25.1211,E2 -310.5621} C_DIS
LIN {X 20.5868,Y 16.4581,Z 61,A 30.3077,B 24.8092,C -3.1852,E1 25.1262,E2 -307.6724} C_DIS
LIN {X 21.5906,Y 15.1172,Z 61,A 26.4407,B 24.8106,C -3.1739,E1 25.1326,E2 -303.7974} C_DIS
LIN {X 22.3499,Y 13.9699,Z 61,A 23.1911,B 24.8118,C -3.1635,E1 25.1375,E2 -300.5395} C_DIS
LIN {X 23.4276,Y 12.076,Z 61,A 18.9625,B 24.8126,C -3.1567,E1 25.1431,E2 -296.317} C_DIS
LIN {X 24.0719,Y 10.7344,Z 61,A 15.5046,B 24.814,C -3.1453,E1 25.1471,E2 -292.8507} C_DIS
LIN {X 24.9339,Y 8.5437,Z 61,A 10.3949,B 24.8157,C -3.1308,E1 25.1521,E2 -287.7352} C_DIS
LIN {X 25.3883,Y 7.0798,Z 61,A 6.2673,B 24.8179,C -3.1118,E1 25.1553,E2 -283.5863} C_DIS
LIN {X 26.0935,Y 3.7155,Z 61,A -0.123,B 24.8191,C -3.1018,E1 25.1585,E2 -277.2095} C_DIS
LIN {X 26.2972,Y 1.7693,Z 61,A -5.0908,B 24.8216,C -3.0803,E1 25.1597,E2 -272.2203} C_DIS
LIN {X 26.3465,Y -0.7377,Z 61,A -9.9566,B 24.8228,C -3.0701,E1 25.1597,E2 -267.3594} C_DIS
LIN {X 26.1976,Y -2.887,Z 61,A -14.1815,B 24.8239,C -3.0609,E1 25.1586,E2 -263.1376} C_DIS
LIN {X 25.9926,Y -4.3657,Z 61,A -17.724,B 24.8255,C -3.0472,E1 25.1571,E2 -259.5836} C_DIS
LIN {X 25.7152,Y -5.7793,Z 61,A -21.0115,B 24.8268,C -3.0357,E1 25.1552,E2 -256.288} C_DIS
LIN {X 25.1343,Y -7.9331,Z 61,A -25.6311,B 24.8282,C -3.0236,E1 25.1516,E2 -251.666} C_DIS
LIN {X 24.6436,Y -9.3473,Z 61,A -28.6825,B 24.829,C -3.0161,E1 25.1487,E2 -248.6142} C_DIS
LIN {X 23.9594,Y -10.9839,Z 61,A -32.6309,B 24.8304,C -3.0037,E1 25.1443,E2 -244.6577} C_DIS
LIN {X 22.8533,Y -13.1302,Z 61,A -37.8561,B 24.8321,C -2.989,E1 25.1374,E2 -239.4252} C_DIS
LIN {X 22.2302,Y -14.1599,Z 61,A -40.5059,B 24.8329,C -2.9813,E1 25.1335,E2 -236.7708} C_DIS
LIN {X 21.2516,Y -15.5899,Z 61,A -43.8504,B 24.8335,C -2.976,E1 25.1281,E2 -233.43} C_DIS
LIN {X 20.6246,Y -16.4104,Z 61,A -46.3568,B 24.8345,C -2.9672,E1 25.1238,E2 -230.9147} C_DIS
LIN {X 19.6692,Y -17.5442,Z 61,A -49.6096,B 24.8355,C -2.9588,E1 25.1178,E2 -227.6565} C_DIS
LIN {X 18.2683,Y -18.9985,Z 61,A -53.6061,B 24.8362,C -2.9527,E1 25.11,E2 -223.6627} C_DIS
LIN {X 17.3306,Y -19.8574,Z 61,A -56.7944,B 24.8374,C -2.9419,E1 25.1033,E2 -220.4613} C_DIS
LIN {X 16.0166,Y -20.9321,Z 61,A -60.2096,B 24.8379,C -2.937,E1 25.0959,E2 -217.0474} C_DIS
LIN {X 15.0214,Y -21.6572,Z 61,A -62.9374,B 24.8386,C -2.9311,E1 25.0896,E2 -214.3151} C_DIS
LIN {X 13.9345,Y -22.372,Z 61,A -66.2787,B 24.8397,C -2.9205,E1 25.0817,E2 -210.9593} C_DIS
LIN {X 11.6995,Y -23.6177,Z 61,A -71.8934,B 24.8408,C -2.9107,E1 25.0679,E2 -205.3373} C_DIS
LIN {X 9.7127,Y -24.5019,Z 61,A -75.8356,B 24.8407,C -2.9119,E1 25.0578,E2 -201.4072} C_DIS
LIN {X 8.3877,Y -24.9863,Z 61,A -79.0916,B 24.8413,C -2.9062,E1 25.0492,E2 -198.1441} C_DIS
LIN {X 6.9006,Y -25.437,Z 61,A -83.0673,B 24.8423,C -2.8967,E1 25.0384,E2 -194.1527} C_DIS
LIN {X 4.4144,Y -25.9845,Z 61,A -88.3388,B 24.8426,C -2.8946,E1 25.024,E2 -188.8825} C_DIS
LIN {X 2.5494,Y -26.2334,Z 61,A -92.5084,B 24.8429,C -2.8915,E1 25.0124,E2 -184.7085} C_DIS
LIN {X 0.4793,Y -26.3523,Z 61,A -96.8289,B 24.8429,C -2.8917,E1 25.0004,E2 -180.3895} C_DIS
LIN {X 0.4793,Y -26.3523,Z 61,A -96.8289,B 24.8429,C -2.8917,E1 25.0004,E2 -180.3895} C_DIS
Enddeposition()
LIN {X 0.1395,Y -25.3702,Z 61,A -95.6731,B 24.8392,C -2.9253,E1 25.0038,E2 -181.6251} C_DIS
Startdeposition()
$VEL.CP = VEL_PRINT
LIN {X 1.9739,Y -25.2948,Z 61,A -91.4372,B 24.8389,C -2.9278,E1 25.0157,E2 -185.8653} C_DIS
LIN {X 4.3644,Y -24.9938,Z 61,A -85.5102,B 24.838,C -2.936,E1 25.0321,E2 -191.8064} C_DIS
LIN {X 5.9108,Y -24.6738,Z 61,A -82.3241,B 24.838,C -2.9357,E1 25.0407,E2 -194.9874} C_DIS
LIN {X 7.458,Y -24.2508,Z 61,A -78.6396,B 24.8375,C -2.9403,E1 25.0506,E2 -198.6764} C_DIS
LIN {X 9.4453,Y -23.5484,Z 61,A -73.9936,B 24.837,C -2.9454,E1 25.0627,E2 -203.3246} C_DIS
LIN {X 11.2801,Y -22.7262,Z 61,A -69.7088,B 24.8365,C -2.9498,E1 25.0735,E2 -207.6088} C_DIS
LIN {X 12.662,Y -21.9862,Z 61,A -66.3138,B 24.836,C -2.9544,E1 25.0818,E2 -211.0047} C_DIS
LIN {X 14.1786,Y -21.0398,Z 61,A -61.5436,B 24.8343,C -2.9697,E1 25.093,E2 -215.7956} C_DIS
LIN {X 16.3128,Y -19.4327,Z 61,A -55.6826,B 24.833,C -2.9806,E1 25.1059,E2 -221.6606} C_DIS
LIN {X 17.814,Y -18.0661,Z 61,A -51.4153,B 24.8322,C -2.9877,E1 25.1145,E2 -225.9273} C_DIS
LIN {X 19.1329,Y -16.6629,Z 61,A -46.7701,B 24.8306,C -3.0018,E1 25.1232,E2 -230.585} C_DIS
LIN {X 20.5399,Y -14.8946,Z 61,A -42.0775,B 24.8297,C -3.0105,E1 25.1311,E2 -235.2761} C_DIS
LIN {X 21.5777,Y -13.3461,Z 61,A -37.815,B 24.8283,C -3.0227,E1 25.1376,E2 -239.546} C_DIS
LIN {X 22.3918,Y -11.93,Z 61,A -34.3358,B 24.8273,C -3.0307,E1 25.1423,E2 -243.0262} C_DIS
LIN {X 23.0579,Y -10.5865,Z 61,A -30.794,B 24.826,C -3.0424,E1 25.1465,E2 -246.5764} C_DIS
LIN {X 23.9436,Y -8.392,Z 61,A -25.0905,B 24.8237,C -3.0626,E1 25.1522,E2 -252.296} C_DIS
LIN {X 24.5706,Y -6.3251,Z 61,A -19.9785,B 24.8216,C -3.0803,E1 25.1559,E2 -257.4206} C_DIS
LIN {X 25.1418,Y -3.4111,Z 61,A -14.16,B 24.8204,C -3.0907,E1 25.1587,E2 -263.2296} C_DIS
LIN {X 25.3138,Y -1.7123,Z 61,A -10.1404,B 24.8188,C -3.1047,E1 25.1596,E2 -267.2585} C_DIS
LIN {X 25.3704,Y 0.1693,Z 61,A -6.0911,B 24.8175,C -3.1156,E1 25.1597,E2 -271.3097} C_DIS
LIN {X 25.294,Y 1.9838,Z 61,A -1.6652,B 24.8155,C -3.1321,E1 25.159,E2 -275.7483} C_DIS
LIN {X 25.0552,Y 3.9949,Z 61,A 2.7992,B 24.814,C -3.1448,E1 25.1572,E2 -280.2166} C_DIS
LIN {X 24.5542,Y 6.3891,Z 61,A 8.1547,B 24.8123,C -3.1594,E1 25.1539,E2 -285.5756} C_DIS
LIN {X 24.0143,Y 8.1879,Z 61,A 12.3867,B 24.8108,C -3.1716,E1 25.1502,E2 -289.8125} C_DIS
LIN {X 23.3293,Y 9.974,Z 61,A 16.9436,B 24.8091,C -3.1865,E1 25.1454,E2 -294.3794} C_DIS
LIN {X 22.3666,Y 11.978,Z 61,A 21.3692,B 24.8082,C -3.1933,E1 25.1399,E2 -298.7977} C_DIS
LIN {X 21.6409,Y 13.2438,Z 61,A 24.9265,B 24.8069,C -3.2047,E1 25.1348,E2 -302.3638} C_DIS
LIN {X 20.6423,Y 14.7519,Z 61,A 29.3006,B 24.8053,C -3.2179,E1 25.1278,E2 -306.7477} C_DIS
LIN {X 19.4961,Y 16.2365,Z 61,A 33.053,B 24.8047,C -3.2224,E1 25.1212,E2 -310.4933} C_DIS
LIN {X 18.4023,Y 17.4668,Z 61,A 36.7862,B 24.8037,C -3.2306,E1 25.1142,E2 -314.2295} C_DIS
LIN {X 17.0466,Y 18.7925,Z 61,A 40.7755,B 24.803,C -3.2361,E1 25.1061,E2 -318.2154} C_DIS
LIN {X 15.9234,Y 19.7528,Z 61,A 44.682,B 24.8016,C -3.2481,E1 25.0977,E2 -322.1355} C_DIS
LIN {X 14.6839,Y 20.6908,Z 61,A 47.7407,B 24.8014,C -3.2494,E1 25.0908,E2 -325.1864} C_DIS
LIN {X 12.5778,Y 22.0347,Z 61,A 54.3581,B 24.7992,C -3.2672,E1 25.0749,E2 -331.8256} C_DIS
LIN {X 10.8045,Y 22.9564,Z 61,A 58.1711,B 24.7994,C -3.2658,E1 25.0654,E2 -335.6251} C_DIS
LIN {X 8.8005,Y 23.7963,Z 61,A 62.746,B 24.7992,C -3.2674,E1 25.0536,E2 -340.1937} C_DIS
LIN {X 7.6842,Y 24.1799,Z 61,A 65.621,B 24.7987,C -3.2715,E1 25.0459,E2 -343.0728} C_DIS
LIN {X 5.8796,Y 24.6814,Z 61,A 69.9377,B 24.7983,C -3.2747,E1 25.0342,E2 -347.3906} C_DIS
LIN {X 4.0471,Y 25.0472,Z 61,A 74.1563,B 24.7981,C -3.2762,E1 25.0227,E2 -351.6082} C_DIS
LIN {X 2.1019,Y 25.2846,Z 61,A 79.1263,B 24.7974,C -3.2814,E1 25.0088,E2 -356.5876} C_DIS
LIN {X -0.5281,Y 25.3662,Z 61,A 84.5218,B 24.7981,C -3.2758,E1 24.9938,E2 -361.9692} C_DIS
LIN {X -2.4226,Y 25.2559,Z 61,A 88.7956,B 24.7984,C -3.2739,E1 24.9819,E2 -366.2402} C_DIS
LIN {X -4.2421,Y 25.0146,Z 61,A 92.9465,B 24.7987,C -3.2712,E1 24.9705,E2 -370.3884} C_DIS
LIN {X -6.3219,Y 24.5714,Z 61,A 97.4826,B 24.7995,C -3.2649,E1 24.9581,E2 -374.9154} C_DIS
LIN {X -7.6724,Y 24.1831,Z 61,A 100.6261,B 24.7999,C -3.2613,E1 24.9498,E2 -378.0555} C_DIS
LIN {X -9.1134,Y 23.6785,Z 61,A 104.4032,B 24.8002,C -3.2593,E1 24.9399,E2 -381.8356} C_DIS
LIN {X -11.1536,Y 22.7888,Z 61,A 109.8703,B 24.8007,C -3.2549,E1 24.926,E2 -387.3057} C_DIS
LIN {X -13.3281,Y 21.589,Z 61,A 114.9394,B 24.8024,C -3.2415,E1 24.9138,E2 -392.3582} C_DIS
LIN {X -14.4959,Y 20.8229,Z 61,A 117.981,B 24.8032,C -3.2348,E1 24.9068,E2 -395.3938} C_DIS
LIN {X -15.5917,Y 20.0159,Z 61,A 121.5445,B 24.8036,C -3.2316,E1 24.8989,E2 -398.9626} C_DIS
LIN {X -16.9972,Y 18.8369,Z 61,A 125.23,B 24.805,C -3.2197,E1 24.8911,E2 -402.634} C_DIS
LIN {X -17.8325,Y 18.0478,Z 61,A 127.7238,B 24.8058,C -3.2131,E1 24.8862,E2 -405.1224} C_DIS
LIN {X -18.6661,Y 17.1843,Z 61,A 130.8922,B 24.8063,C -3.2093,E1 24.8801,E2 -408.2957} C_DIS
LIN {X -19.8596,Y 15.7899,Z 61,A 135.0069,B 24.8076,C -3.1986,E1 24.8728,E2 -412.4038} C_DIS
LIN {X -20.7152,Y 14.6497,Z 61,A 138.2965,B 24.8086,C -3.1905,E1 24.8675,E2 -415.6901} C_DIS
LIN {X -21.9662,Y 12.6969,Z 61,A 143.6278,B 24.8102,C -3.1766,E1 24.8597,E2 -421.0153} C_DIS
LIN {X -22.6348,Y 11.4629,Z 61,A 146.7517,B 24.8114,C -3.1673,E1 24.8557,E2 -424.1336} C_DIS
LIN {X -23.3728,Y 9.8709,Z 61,A 150.8109,B 24.8127,C -3.1562,E1 24.8512,E2 -428.1886} C_DIS
LIN {X -24.0465,Y 8.0914,Z 61,A 155.887,B 24.8137,C -3.1476,E1 24.8465,E2 -433.2729} C_DIS
LIN {X -24.8891,Y 4.9267,Z 61,A 162.4189,B 24.817,C -3.1201,E1 24.8423,E2 -439.7772} C_DIS
LIN {X -25.194,Y 2.998,Z 61,A 167.0792,B 24.8184,C -3.1077,E1 24.8405,E2 -444.4356} C_DIS
LIN {X -25.3594,Y 0.7894,Z 61,A 171.9482,B 24.8203,C -3.0914,E1 24.8398,E2 -449.2948} C_DIS
LIN {X -25.3532,Y -0.9757,Z 61,A 175.5622,B 24.822,C -3.077,E1 24.84,E2 -452.8961} C_DIS
LIN {X -25.2775,Y -2.1822,Z 61,A 178.5239,B 24.8228,C -3.0698,E1 24.8406,E2 -455.8584} C_DIS
LIN {X -25.1076,Y -3.6516,Z 61,A -177.8915,B 24.8239,C -3.0609,E1 24.8419,E2 -459.4431} C_DIS
LIN {X -24.7642,Y -5.5199,Z 61,A -173.6026,B 24.8254,C -3.048,E1 24.8443,E2 -463.7263} C_DIS
LIN {X -24.2903,Y -7.3291,Z 61,A -169.292,B 24.8267,C -3.036,E1 24.8476,E2 -468.0333} C_DIS
LIN {X -23.4907,Y -9.587,Z 61,A -163.5815,B 24.8283,C -3.0224,E1 24.8532,E2 -473.7432} C_DIS
LIN {X -22.746,Y -11.2402,Z 61,A -159.4094,B 24.8295,C -3.0117,E1 24.8583,E2 -477.9124} C_DIS
LIN {X -21.5862,Y -13.3332,Z 61,A -154.8322,B 24.8317,C -2.9928,E1 24.8646,E2 -482.4683} C_DIS
LIN {X -20.7921,Y -14.5402,Z 61,A -150.7087,B 24.832,C -2.9901,E1 24.8712,E2 -486.6055} C_DIS
LIN {X -19.4976,Y -16.2347,Z 61,A -146.481,B 24.8336,C -2.9753,E1 24.8785,E2 -490.8177} C_DIS
LIN {X -18.4471,Y -17.4193,Z 61,A -142.5998,B 24.8343,C -2.9696,E1 24.8858,E2 -494.7024} C_DIS
LIN {X -16.728,Y -19.0761,Z 61,A -137.4885,B 24.8357,C -2.9571,E1 24.8962,E2 -499.8048} C_DIS
LIN {X -14.9331,Y -20.5117,Z 61,A -131.3711,B 24.836,C -2.9545,E1 24.9098,E2 -505.9382} C_DIS
LIN {X -13.4619,Y -21.5058,Z 61,A -127.9736,B 24.8371,C -2.9442,E1 24.9178,E2 -509.322} C_DIS
LIN {X -11.6849,Y -22.5205,Z 61,A -123.6951,B 24.838,C -2.9357,E1 24.9282,E2 -513.5924} C_DIS
LIN {X -10.6787,Y -23.015,Z 61,A -121.1043,B 24.8383,C -2.9332,E1 24.9348,E2 -516.1839} C_DIS
LIN {X -9.549,Y -23.5061,Z 61,A -117.9894,B 24.8383,C -2.933,E1 24.9428,E2 -519.3054} C_DIS
LIN {X -7.7609,Y -24.1556,Z 61,A -113.7571,B 24.8388,C -2.9291,E1 24.954,E2 -523.5364} C_DIS
LIN {X -5.9783,Y -24.6573,Z 61,A -109.5188,B 24.839,C -2.9271,E1 24.9654,E2 -527.7763} C_DIS
LIN {X -3.8713,Y -25.0743,Z 61,A -104.8551,B 24.8393,C -2.924,E1 24.9782,E2 -532.4373} C_DIS
LIN {X -2.3427,Y -25.263,Z 61,A -101.1102,B 24.8391,C -2.9259,E1 24.9887,E2 -536.1889} C_DIS
LIN {X -0.8604,Y -25.3572,Z 61,A -97.8276,B 24.8391,C -2.9256,E1 24.9978,E2 -539.4715} C_DIS
LIN {X -0.8604,Y -25.3572,Z 61,A -97.8276,B 24.8391,C -2.9256,E1 24.9978,E2 -539.4715} C_DIS
Enddeposition()
LIN {X 0.1346,Y -24.3815,Z 61,A -96.6732,B 24.8383,C -2.9336,E1 25.0011,E2 -540.645} C_DIS
Startdeposition()
$VEL.CP = VEL_PRINT
LIN {X -1.2943,Y -24.3523,Z 61,A -101.2868,B 24.8395,C -2.9229,E1 24.9882,E2 -536.0052} C_DIS
LIN {X -3.5926,Y -24.1209,Z 61,A -106.4838,B 24.8392,C -2.9256,E1 24.9738,E2 -530.8109} C_DIS
LIN {X -5.3567,Y -23.7914,Z 61,A -110.6239,B 24.8389,C -2.9278,E1 24.9624,E2 -526.6714} C_DIS
LIN {X -7.0566,Y -23.3437,Z 61,A -114.8537,B 24.8387,C -2.9297,E1 24.9511,E2 -522.4393} C_DIS
LIN {X -8.8154,Y -22.7378,Z 61,A -119.2369,B 24.8383,C -2.9334,E1 24.9396,E2 -518.056} C_DIS
LIN {X -10.2924,Y -22.1082,Z 61,A -122.6111,B 24.8376,C -2.9401,E1 24.931,E2 -514.6898} C_DIS
LIN {X -11.7571,Y -21.3659,Z 61,A -126.9006,B 24.8373,C -2.9421,E1 24.9204,E2 -510.393} C_DIS
LIN {X -12.9901,Y -20.6391,Z 61,A -130.124,B 24.8367,C -2.9478,E1 24.9127,E2 -507.1733} C_DIS
LIN {X -14.5271,Y -19.5881,Z 61,A -134.7188,B 24.8361,C -2.9535,E1 24.9022,E2 -502.5763} C_DIS
LIN {X -15.9967,Y -18.407,Z 61,A -138.8665,B 24.835,C -2.9633,E1 24.8934,E2 -498.4363} C_DIS
LIN {X -17.2894,Y -17.1987,Z 61,A -143.3048,B 24.8342,C -2.97,E1 24.8844,E2 -493.9955} C_DIS
LIN {X -18.5643,Y -15.8138,Z 61,A -148.0521,B 24.8333,C -2.9779,E1 24.8757,E2 -489.2456} C_DIS
LIN {X -19.8662,Y -14.1436,Z 61,A -152.7179,B 24.8318,C -2.9914,E1 24.8679,E2 -484.5896} C_DIS
LIN {X -20.8675,Y -12.6199,Z 61,A -157.084,B 24.8306,C -3.0017,E1 24.8614,E2 -480.2261} C_DIS
LIN {X -21.97,Y -10.5844,Z 61,A -162.2264,B 24.8288,C -3.0178,E1 24.8548,E2 -475.0947} C_DIS
LIN {X -22.7539,Y -8.7744,Z 61,A -167.2252,B 24.8276,C -3.0289,E1 24.8495,E2 -470.0947} C_DIS
LIN {X -23.3711,Y -6.9644,Z 61,A -171.6727,B 24.826,C -3.0421,E1 24.8457,E2 -465.6535} C_DIS
LIN {X -23.8198,Y -5.2276,Z 61,A -175.8989,B 24.8246,C -3.0547,E1 24.8429,E2 -461.4325} C_DIS
LIN {X -24.1407,Y -3.455,Z 61,A 179.787,B 24.8232,C -3.0671,E1 24.841,E2 -457.1227} C_DIS
LIN {X -24.2989,Y -2.0714,Z 61,A 176.7069,B 24.8219,C -3.0781,E1 24.8402,E2 -454.0504} C_DIS
LIN {X -24.382,Y -0.4768,Z 61,A 172.5668,B 24.8207,C -3.0879,E1 24.8398,E2 -449.9088} C_DIS
LIN {X -24.3478,Y 1.3719,Z 61,A 168.9036,B 24.8188,C -3.1047,E1 24.8401,E2 -446.2639} C_DIS
LIN {X -24.2144,Y 2.8936,Z 61,A 164.4911,B 24.8179,C -3.112,E1 24.8414,E2 -441.8423} C_DIS
LIN {X -23.9192,Y 4.7536,Z 61,A 160.0973,B 24.8163,C -3.1259,E1 24.8436,E2 -437.4557} C_DIS
LIN {X -23.3248,Y 7.1187,Z 61,A 154.4228,B 24.8142,C -3.1437,E1 24.8477,E2 -431.7909} C_DIS
LIN {X -22.6988,Y 8.9147,Z 61,A 149.9811,B 24.8126,C -3.1571,E1 24.852,E2 -427.3564} C_DIS
LIN {X -21.9421,Y 10.6423,Z 61,A 145.7698,B 24.8109,C -3.1711,E1 24.8569,E2 -423.1557} C_DIS
LIN {X -21.2872,Y 11.8982,Z 61,A 142.6722,B 24.8096,C -3.1817,E1 24.861,E2 -420.0671} C_DIS
LIN {X -20.5597,Y 13.1153,Z 61,A 138.802,B 24.8088,C -3.1882,E1 24.8667,E2 -416.1924} C_DIS
LIN {X -19.4963,Y 14.6494,Z 61,A 134.6121,B 24.8073,C -3.2008,E1 24.8735,E2 -412.0123} C_DIS
LIN {X -18.4341,Y 15.9657,Z 61,A 130.3595,B 24.8063,C -3.2093,E1 24.8811,E2 -407.7606} C_DIS
LIN {X -17.1892,Y 17.2987,Z 61,A 125.5535,B 24.8054,C -3.2166,E1 24.8905,E2 -402.9515} C_DIS
LIN {X -15.4335,Y 18.8819,Z 61,A 120.7999,B 24.8034,C -3.2332,E1 24.9005,E2 -398.2191} C_DIS
LIN {X -13.8465,Y 20.0743,Z 61,A 115.5659,B 24.8027,C -3.2391,E1 24.9123,E2 -392.9809} C_DIS
LIN {X -12.1515,Y 21.1436,Z 61,A 110.4983,B 24.8019,C -3.2453,E1 24.9245,E2 -387.9125} C_DIS
LIN {X -9.2597,Y 22.5604,Z 61,A 102.9326,B 24.8005,C -3.2564,E1 24.9437,E2 -380.3549} C_DIS
LIN {X -6.5739,Y 23.484,Z 61,A 96.8333,B 24.7991,C -3.2677,E1 24.9599,E2 -374.2718} C_DIS
LIN {X -4.7518,Y 23.9197,Z 61,A 92.3119,B 24.7988,C -3.2706,E1 24.9722,E2 -369.7517} C_DIS
LIN {X -2.8438,Y 24.2203,Z 61,A 87.8044,B 24.7984,C -3.2737,E1 24.9847,E2 -365.248} C_DIS
LIN {X -1.3306,Y 24.3503,Z 61,A 84.7845,B 24.7977,C -3.2792,E1 24.993,E2 -362.2401} C_DIS
Enddeposition()
END
